LIN {X 0,Y 474.683,Z 210.352,A -85,B 0,C 180,E1 -7368.037,E2 -7368.037} C_VEL
LIN {X 0,Y 474.691,Z 210.355,A -85,B 0,C 180,E1 -7371.486,E2 -7371.486} C_VEL
LIN {X 0,Y 474.74,Z 210.345,A -85,B 0,C 180,E1 -7374.052,E2 -7374.052} C_VEL
LIN {X 0,Y 474.841,Z 210.335,A -85,B 0,C 180,E1 -7377.455,E2 -7377.455} C_VEL
LIN {X 0,Y 474.818,Z 210.341,A -85,B 0,C 180,E1 -7380.848,E2 -7380.848} C_VEL
LIN {X 0,Y 474.835,Z 210.335,A -85,B 0,C 180,E1 -7382.545,E2 -7382.545} C_VEL
LIN {X 0,Y 474.723,Z 210.347,A -85,B 0,C 180,E1 -7385.948,E2 -7385.948} C_VEL
LIN {X 0,Y 474.671,Z 210.356,A -85,B 0,C 180,E1 -7388.515,E2 -7388.515} C_VEL
LIN {X 0,Y 474.683,Z 210.352,A -85,B 0,C 180,E1 -7391.963,E2 -7391.963} C_VEL
LIN {X 0,Y 474.647,Z 210.356,A -85,B 0,C 180,E1 -7395.779,E2 -7395.779} C_VEL
LIN {X 0,Y 474.611,Z 210.365,A -85,B 0,C 180,E1 -7399.013,E2 -7399.013} C_VEL
LIN {X 0,Y 474.545,Z 210.369,A -85,B 0,C 180,E1 -7401.731,E2 -7401.731} C_VEL
LIN {X 0,Y 474.611,Z 210.367,A -85,B 0,C 180,E1 -7404.496,E2 -7404.496} C_VEL
LIN {X 0,Y 474.652,Z 210.356,A -85,B 0,C 180,E1 -7407.342,E2 -7407.342} C_VEL
LIN {X 0,Y 474.565,Z 210.371,A -85,B 0,C 180,E1 -7410.815,E2 -7410.815} C_VEL
LIN {X 0,Y 474.597,Z 210.365,A -85,B 0,C 180,E1 -7413.988,E2 -7413.988} C_VEL
LIN {X 0,Y 474.534,Z 210.372,A -85,B 0,C 180,E1 -7416.903,E2 -7416.903} C_VEL
LIN {X 0,Y 474.611,Z 210.362,A -85,B 0,C 180,E1 -7419.654,E2 -7419.654} C_VEL
LIN {X 0,Y 474.618,Z 210.361,A -85,B 0,C 180,E1 -7422.934,E2 -7422.934} C_VEL
LIN {X 0,Y 474.579,Z 210.368,A -85,B 0,C 180,E1 -7425.899,E2 -7425.899} C_VEL
LIN {X 0,Y 474.601,Z 210.362,A -85,B 0,C 180,E1 -7429.045,E2 -7429.045} C_VEL
LIN {X 0,Y 474.586,Z 210.367,A -85,B 0,C 180,E1 -7431.708,E2 -7431.708} C_VEL
LIN {X 0,Y 474.608,Z 210.362,A -85,B 0,C 180,E1 -7434.73,E2 -7434.73} C_VEL
LIN {X 0,Y 474.617,Z 210.365,A -85,B 0,C 180,E1 -7437.792,E2 -7437.792} C_VEL
LIN {X 0,Y 474.608,Z 210.361,A -85,B 0,C 180,E1 -7440.889,E2 -7440.889} C_VEL
LIN {X 0,Y 474.642,Z 210.361,A -85,B 0,C 180,E1 -7443.632,E2 -7443.632} C_VEL
LIN {X 0,Y 474.625,Z 210.359,A -85,B 0,C 180,E1 -7446.645,E2 -7446.645} C_VEL
LIN {X 0,Y 474.646,Z 210.361,A -85,B 0,C 180,E1 -7450.093,E2 -7450.093} C_VEL
LIN {X 0,Y 474.638,Z 210.362,A -85,B 0,C 180,E1 -7451.71,E2 -7451.71} C_VEL
LIN {X 0,Y 473.972,Z 210.45,A -85,B 0,C 180,E1 -7452.419,E2 -7452.419} C_VEL
LIN {X 0,Y 471.122,Z 210.804,A -85,B 0,C 180,E1 -7453.571,E2 -7453.571} C_VEL
LIN {X 0,Y 468.711,Z 211.1,A -85,B 0,C 180,E1 -7454.5,E2 -7454.5} C_VEL
LIN {X 0,Y 467.673,Z 211.227,A -85,B 0,C 180,E1 -7455.217,E2 -7455.217} C_VEL
LIN {X 0,Y 467.588,Z 211.236,A -85,B 0,C 180,E1 -7455.46,E2 -7455.46} C_VEL
LIN {X 0,Y 467.65,Z 211.232,A -85,B 0,C 180,E1 -7458.737,E2 -7458.737} C_VEL
LIN {X 0,Y 467.708,Z 211.37,A -85,B 0,C 180,E1 -7461.142,E2 -7461.142} C_VEL
LIN {X 0,Y 468.579,Z 217.66,A -85,B 0,C 180,E1 -7462.461,E2 -7462.461} C_VEL
LIN {X 0,Y 468.348,Z 226.062,A -85,B 0,C 180,E1 -7464.135,E2 -7464.135} C_VEL
LIN {X 0,Y 471.304,Z 240.96,A -85,B 0,C 180,E1 -7464.467,E2 -7464.467} C_VEL
LIN {X 0,Y 470.437,Z 333.788,A -85,B 0,C 180,E1 -7465.906,E2 -7465.906} C_VEL
LIN {X 0,Y 470.197,Z 347.368,A -85,B 0,C 180,E1 -7466.306,E2 -7466.306} C_VEL
LIN {X 0,Y 469.865,Z 359.62,A -85,B 0,C 180,E1 -7466.84,E2 -7466.84} C_VEL
LIN {X 0,Y 469.485,Z 371.367,A -85,B 0,C 180,E1 -7467.535,E2 -7467.535} C_VEL
LIN {X 0,Y 468.946,Z 382.682,A -85,B 0,C 180,E1 -7468.392,E2 -7468.392} C_VEL
LIN {X 0,Y 468.486,Z 392.879,A -85,B 0,C 180,E1 -7469.357,E2 -7469.357} C_VEL
LIN {X 0,Y 468.059,Z 402.058,A -85,B 0,C 180,E1 -7470.432,E2 -7470.432} C_VEL
LIN {X 0,Y 467.627,Z 410.968,A -85,B 0,C 180,E1 -7471.724,E2 -7471.724} C_VEL
LIN {X 0,Y 467.285,Z 418.164,A -85,B 0,C 180,E1 -7473.019,E2 -7473.019} C_VEL
LIN {X 0,Y 467.131,Z 423.923,A -85,B 0,C 180,E1 -7474.315,E2 -7474.315} C_VEL
LIN {X 0,Y 466.93,Z 428.479,A -85,B 0,C 180,E1 -7475.616,E2 -7475.616} C_VEL
LIN {X 0,Y 466.819,Z 431.951,A -85,B 0,C 180,E1 -7476.918,E2 -7476.918} C_VEL
LIN {X 0,Y 466.739,Z 433.696,A -85,B 0,C 180,E1 -7477.79,E2 -7477.79} C_VEL
LIN {X 0,Y 466.615,Z 435.959,A -85,B 0,C 180,E1 -7479.537,E2 -7479.537} C_VEL
LIN {X 0,Y 466.637,Z 436.49,A -85,B 0,C 180,E1 -7480.413,E2 -7480.413} C_VEL
LIN {X 0,Y 466.688,Z 436.48,A -85,B 0,C 180,E1 -7481.802,E2 -7481.802} C_VEL
LIN {X 0,Y 466.63,Z 435.592,A -85,B 0,C 180,E1 -7483.057,E2 -7483.057} C_VEL
LIN {X 0,Y 466.66,Z 434.468,A -85,B 0,C 180,E1 -7483.944,E2 -7483.944} C_VEL
LIN {X 0,Y 466.848,Z 431.331,A -85,B 0,C 180,E1 -7485.534,E2 -7485.534} C_VEL
LIN {X 0,Y 466.999,Z 426.929,A -85,B 0,C 180,E1 -7487.065,E2 -7487.065} C_VEL
LIN {X 0,Y 467.242,Z 421.768,A -85,B 0,C 180,E1 -7488.413,E2 -7488.413} C_VEL
LIN {X 0,Y 467.513,Z 415.168,A -85,B 0,C 180,E1 -7489.769,E2 -7489.769} C_VEL
LIN {X 0,Y 468.017,Z 406.854,A -85,B 0,C 180,E1 -7491.124,E2 -7491.124} C_VEL
LIN {X 0,Y 468.456,Z 398.271,A -85,B 0,C 180,E1 -7492.26,E2 -7492.26} C_VEL
LIN {X 0,Y 468.921,Z 388.788,A -85,B 0,C 180,E1 -7493.284,E2 -7493.284} C_VEL
LIN {X 0,Y 469.432,Z 378.914,A -85,B 0,C 180,E1 -7494.148,E2 -7494.148} C_VEL
LIN {X 0,Y 469.92,Z 366.789,A -85,B 0,C 180,E1 -7494.992,E2 -7494.992} C_VEL
LIN {X 0,Y 470.292,Z 354.995,A -85,B 0,C 180,E1 -7495.622,E2 -7495.622} C_VEL
LIN {X 0,Y 470.657,Z 341.985,A -85,B 0,C 180,E1 -7496.114,E2 -7496.114} C_VEL
LIN {X 0,Y 470.883,Z 328.515,A -85,B 0,C 180,E1 -7496.434,E2 -7496.434} C_VEL
LIN {X 0,Y 471.54,Z 239.78,A -85,B 0,C 180,E1 -7497.811,E2 -7497.811} C_VEL
LIN {X 0,Y 468.611,Z 226.016,A -85,B 0,C 180,E1 -7498.174,E2 -7498.174} C_VEL
LIN {X 0,Y 468.575,Z 216.184,A -85,B 0,C 180,E1 -7500.161,E2 -7500.161} C_VEL
LIN {X 0,Y 467.602,Z 211.238,A -85,B 0,C 180,E1 -7501.263,E2 -7501.263} C_VEL
LIN {X 0,Y 467.585,Z 211.242,A -85,B 0,C 180,E1 -7504.241,E2 -7504.241} C_VEL
LIN {X 0,Y 467.544,Z 211.246,A -85,B 0,C 180,E1 -7507.185,E2 -7507.185} C_VEL
LIN {X 0,Y 467.586,Z 211.241,A -85,B 0,C 180,E1 -7510.261,E2 -7510.261} C_VEL
LIN {X 0,Y 467.577,Z 211.243,A -85,B 0,C 180,E1 -7512.565,E2 -7512.565} C_VEL
LIN {X 0,Y 467.562,Z 211.248,A -85,B 0,C 180,E1 -7516.175,E2 -7516.175} C_VEL
LIN {X 0,Y 467.575,Z 211.24,A -85,B 0,C 180,E1 -7518.72,E2 -7518.72} C_VEL
LIN {X 0,Y 467.552,Z 211.247,A -85,B 0,C 180,E1 -7521.954,E2 -7521.954} C_VEL
LIN {X 0,Y 467.548,Z 211.241,A -85,B 0,C 180,E1 -7525.166,E2 -7525.166} C_VEL
LIN {X 0,Y 467.563,Z 211.24,A -85,B 0,C 180,E1 -7528.258,E2 -7528.258} C_VEL
LIN {X 0,Y 467.558,Z 211.242,A -85,B 0,C 180,E1 -7531.249,E2 -7531.249} C_VEL
LIN {X 0,Y 467.586,Z 211.24,A -85,B 0,C 180,E1 -7534.158,E2 -7534.158} C_VEL
LIN {X 0,Y 467.553,Z 211.238,A -85,B 0,C 180,E1 -7536.994,E2 -7536.994} C_VEL
LIN {X 0,Y 467.595,Z 211.237,A -85,B 0,C 180,E1 -7539.776,E2 -7539.776} C_VEL
LIN {X 0,Y 467.583,Z 211.237,A -85,B 0,C 180,E1 -7542.506,E2 -7542.506} C_VEL
LIN {X 0,Y 467.575,Z 211.238,A -85,B 0,C 180,E1 -7545.195,E2 -7545.195} C_VEL
LIN {X 0,Y 467.625,Z 211.233,A -85,B 0,C 180,E1 -7547.854,E2 -7547.854} C_VEL
LIN {X 0,Y 467.651,Z 211.236,A -85,B 0,C 180,E1 -7551.357,E2 -7551.357} C_VEL
LIN {X 0,Y 467.723,Z 211.218,A -85,B 0,C 180,E1 -7553.962,E2 -7553.962} C_VEL
LIN {X 0,Y 467.825,Z 211.208,A -85,B 0,C 180,E1 -7557.417,E2 -7557.417} C_VEL
LIN {X 0,Y 467.844,Z 211.204,A -85,B 0,C 180,E1 -7560,E2 -7560} C_VEL
LIN {X 0,Y 467.823,Z 211.206,A -85,B 0,C 180,E1 -7562.583,E2 -7562.583} C_VEL
LIN {X 0,Y 467.695,Z 211.222,A -85,B 0,C 180,E1 -7566.038,E2 -7566.038} C_VEL
LIN {X 0,Y 467.638,Z 211.229,A -85,B 0,C 180,E1 -7568.644,E2 -7568.644} C_VEL
LIN {X 0,Y 467.643,Z 211.226,A -85,B 0,C 180,E1 -7572.146,E2 -7572.146} C_VEL
LIN {X 0,Y 467.618,Z 211.231,A -85,B 0,C 180,E1 -7575.885,E2 -7575.885} C_VEL
LIN {X 0,Y 467.592,Z 211.238,A -85,B 0,C 180,E1 -7579.309,E2 -7579.309} C_VEL
LIN {X 0,Y 467.502,Z 211.244,A -85,B 0,C 180,E1 -7582.075,E2 -7582.075} C_VEL
LIN {X 0,Y 467.543,Z 211.243,A -85,B 0,C 180,E1 -7584.891,E2 -7584.891} C_VEL
LIN {X 0,Y 467.555,Z 211.241,A -85,B 0,C 180,E1 -7587.773,E2 -7587.773} C_VEL
LIN {X 0,Y 467.527,Z 211.246,A -85,B 0,C 180,E1 -7591.042,E2 -7591.042} C_VEL
LIN {X 0,Y 467.555,Z 211.242,A -85,B 0,C 180,E1 -7594.242,E2 -7594.242} C_VEL
LIN {X 0,Y 467.526,Z 211.239,A -85,B 0,C 180,E1 -7597.187,E2 -7597.187} C_VEL
LIN {X 0,Y 467.555,Z 211.241,A -85,B 0,C 180,E1 -7600.267,E2 -7600.267} C_VEL
LIN {X 0,Y 467.572,Z 211.242,A -85,B 0,C 180,E1 -7602.569,E2 -7602.569} C_VEL
LIN {X 0,Y 467.551,Z 211.24,A -85,B 0,C 180,E1 -7605.054,E2 -7605.054} C_VEL
LIN {X 0,Y 467.555,Z 211.242,A -85,B 0,C 180,E1 -7608.598,E2 -7608.598} C_VEL
LIN {X 0,Y 467.554,Z 211.243,A -85,B 0,C 180,E1 -7611.957,E2 -7611.957} C_VEL
LIN {X 0,Y 467.558,Z 211.241,A -85,B 0,C 180,E1 -7615.169,E2 -7615.169} C_VEL
LIN {X 0,Y 467.578,Z 211.244,A -85,B 0,C 180,E1 -7618.261,E2 -7618.261} C_VEL
LIN {X 0,Y 467.552,Z 211.245,A -85,B 0,C 180,E1 -7621.25,E2 -7621.25} C_VEL
LIN {X 0,Y 467.622,Z 211.273,A -85,B 0,C 180,E1 -7623.352,E2 -7623.352} C_VEL
LIN {X 0,Y 469.977,Z 223.105,A -85,B 0,C 180,E1 -7625.581,E2 -7625.581} C_VEL
LIN {X 0,Y 469.825,Z 230.597,A -85,B 0,C 180,E1 -7626.88,E2 -7626.88} C_VEL
LIN {X 0,Y 469.021,Z 248.029,A -85,B 0,C 180,E1 -7629.84,E2 -7629.84} C_VEL
LIN {X 0,Y 468.331,Z 266.089,A -85,B 0,C 180,E1 -7632.866,E2 -7632.866} C_VEL
LIN {X 0,Y 471.36,Z 286.814,A -85,B 0,C 180,E1 -7633.329,E2 -7633.329} C_VEL
LIN {X 0,Y 470.641,Z 375.192,A -85,B 0,C 180,E1 -7634.713,E2 -7634.713} C_VEL
LIN {X 0,Y 470.204,Z 389.075,A -85,B 0,C 180,E1 -7635.114,E2 -7635.114} C_VEL
LIN {X 0,Y 469.721,Z 401.519,A -85,B 0,C 180,E1 -7635.652,E2 -7635.652} C_VEL
LIN {X 0,Y 469.208,Z 413.424,A -85,B 0,C 180,E1 -7636.354,E2 -7636.354} C_VEL
LIN {X 0,Y 468.662,Z 425.211,A -85,B 0,C 180,E1 -7637.25,E2 -7637.25} C_VEL
LIN {X 0,Y 468.137,Z 436.204,A -85,B 0,C 180,E1 -7638.306,E2 -7638.306} C_VEL
LIN {X 0,Y 467.673,Z 445.316,A -85,B 0,C 180,E1 -7639.391,E2 -7639.391} C_VEL
LIN {X 0,Y 467.248,Z 454.216,A -85,B 0,C 180,E1 -7640.694,E2 -7640.694} C_VEL
LIN {X 0,Y 466.987,Z 461.379,A -85,B 0,C 180,E1 -7641.997,E2 -7641.997} C_VEL
LIN {X 0,Y 466.831,Z 466.228,A -85,B 0,C 180,E1 -7643.082,E2 -7643.082} C_VEL
LIN {X 0,Y 466.733,Z 470.943,A -85,B 0,C 180,E1 -7644.382,E2 -7644.382} C_VEL
LIN {X 0,Y 466.648,Z 474.545,A -85,B 0,C 180,E1 -7645.68,E2 -7645.68} C_VEL
LIN {X 0,Y 466.691,Z 476.404,A -85,B 0,C 180,E1 -7646.545,E2 -7646.545} C_VEL
LIN {X 0,Y 466.68,Z 477.796,A -85,B 0,C 180,E1 -7647.409,E2 -7647.409} C_VEL
LIN {X 0,Y 466.661,Z 478.792,A -85,B 0,C 180,E1 -7648.273,E2 -7648.273} C_VEL
LIN {X 0,Y 466.624,Z 479.396,A -85,B 0,C 180,E1 -7649.135,E2 -7649.135} C_VEL
LIN {X 0,Y 466.607,Z 479.602,A -85,B 0,C 180,E1 -7649.998,E2 -7649.998} C_VEL
LIN {X 0,Y 466.661,Z 478.761,A -85,B 0,C 180,E1 -7651.724,E2 -7651.724} C_VEL
LIN {X 0,Y 466.679,Z 477.755,A -85,B 0,C 180,E1 -7652.588,E2 -7652.588} C_VEL
LIN {X 0,Y 466.691,Z 476.337,A -85,B 0,C 180,E1 -7653.451,E2 -7653.451} C_VEL
LIN {X 0,Y 466.687,Z 473.368,A -85,B 0,C 180,E1 -7654.749,E2 -7654.749} C_VEL
LIN {X 0,Y 466.743,Z 469.348,A -85,B 0,C 180,E1 -7656.048,E2 -7656.048} C_VEL
LIN {X 0,Y 466.906,Z 463.158,A -85,B 0,C 180,E1 -7657.566,E2 -7657.566} C_VEL
LIN {X 0,Y 467.121,Z 456.401,A -85,B 0,C 180,E1 -7658.869,E2 -7658.869} C_VEL
LIN {X 0,Y 467.448,Z 448.015,A -85,B 0,C 180,E1 -7660.173,E2 -7660.173} C_VEL
LIN {X 0,Y 467.905,Z 439.387,A -85,B 0,C 180,E1 -7661.257,E2 -7661.257} C_VEL
LIN {X 0,Y 468.333,Z 429.269,A -85,B 0,C 180,E1 -7662.295,E2 -7662.295} C_VEL
LIN {X 0,Y 468.864,Z 418.178,A -85,B 0,C 180,E1 -7663.211,E2 -7663.211} C_VEL
LIN {X 0,Y 469.352,Z 406.508,A -85,B 0,C 180,E1 -7663.969,E2 -7663.969} C_VEL
LIN {X 0,Y 469.8,Z 394.374,A -85,B 0,C 180,E1 -7664.564,E2 -7664.564} C_VEL
LIN {X 0,Y 470.189,Z 381.179,A -85,B 0,C 180,E1 -7665.022,E2 -7665.022} C_VEL
LIN {X 0,Y 470.523,Z 368.479,A -85,B 0,C 180,E1 -7665.288,E2 -7665.288} C_VEL
LIN {X 0,Y 470.883,Z 285.054,A -85,B 0,C 180,E1 -7666.568,E2 -7666.568} C_VEL
LIN {X 0,Y 468.204,Z 266.3,A -85,B 0,C 180,E1 -7666.966,E2 -7666.966} C_VEL
LIN {X 0,Y 468.844,Z 248.358,A -85,B 0,C 180,E1 -7669.936,E2 -7669.936} C_VEL
LIN {X 0,Y 469.498,Z 230.626,A -85,B 0,C 180,E1 -7672.9,E2 -7672.9} C_VEL
LIN {X 0,Y 469.801,Z 223.259,A -85,B 0,C 180,E1 -7674.142,E2 -7674.142} C_VEL
LIN {X 0,Y 467.665,Z 211.233,A -85,B 0,C 180,E1 -7676.311,E2 -7676.311} C_VEL
LIN {X 0,Y 467.554,Z 211.243,A -85,B 0,C 180,E1 -7679.329,E2 -7679.329} C_VEL
LIN {X 0,Y 467.563,Z 211.24,A -85,B 0,C 180,E1 -7682.675,E2 -7682.675} C_VEL
LIN {X 0,Y 467.541,Z 211.246,A -85,B 0,C 180,E1 -7685.736,E2 -7685.736} C_VEL
LIN {X 0,Y 467.556,Z 211.24,A -85,B 0,C 180,E1 -7689.141,E2 -7689.141} C_VEL
LIN {X 0,Y 467.558,Z 211.24,A -85,B 0,C 180,E1 -7692.563,E2 -7692.563} C_VEL
LIN {X 0,Y 467.541,Z 211.245,A -85,B 0,C 180,E1 -7696.173,E2 -7696.173} C_VEL
LIN {X 0,Y 467.556,Z 211.24,A -85,B 0,C 180,E1 -7698.718,E2 -7698.718} C_VEL
LIN {X 0,Y 467.541,Z 211.245,A -85,B 0,C 180,E1 -7701.403,E2 -7701.403} C_VEL
LIN {X 0,Y 467.522,Z 211.245,A -85,B 0,C 180,E1 -7704.257,E2 -7704.257} C_VEL
LIN {X 0,Y 467.54,Z 211.246,A -85,B 0,C 180,E1 -7707.317,E2 -7707.317} C_VEL
LIN {X 0,Y 467.532,Z 211.243,A -85,B 0,C 180,E1 -7710.663,E2 -7710.663} C_VEL
LIN {X 0,Y 467.572,Z 211.242,A -85,B 0,C 180,E1 -7713.197,E2 -7713.197} C_VEL
LIN {X 0,Y 467.537,Z 211.243,A -85,B 0,C 180,E1 -7716.055,E2 -7716.055} C_VEL
LIN {X 0,Y 467.605,Z 211.235,A -85,B 0,C 180,E1 -7718.856,E2 -7718.856} C_VEL
LIN {X 0,Y 467.58,Z 211.242,A -85,B 0,C 180,E1 -7721.6,E2 -7721.6} C_VEL
LIN {X 0,Y 467.6,Z 211.234,A -85,B 0,C 180,E1 -7724.304,E2 -7724.304} C_VEL
LIN {X 0,Y 467.641,Z 211.23,A -85,B 0,C 180,E1 -7727.854,E2 -7727.854} C_VEL
LIN {X 0,Y 467.64,Z 211.235,A -85,B 0,C 180,E1 -7731.357,E2 -7731.357} C_VEL
LIN {X 0,Y 467.704,Z 211.221,A -85,B 0,C 180,E1 -7733.962,E2 -7733.962} C_VEL
LIN {X 0,Y 467.808,Z 211.212,A -85,B 0,C 180,E1 -7737.417,E2 -7737.417} C_VEL
LIN {X 0,Y 467.77,Z 211.219,A -85,B 0,C 180,E1 -7740.861,E2 -7740.861} C_VEL
LIN {X 0,Y 467.801,Z 211.212,A -85,B 0,C 180,E1 -7742.583,E2 -7742.583} C_VEL
LIN {X 0,Y 467.687,Z 211.223,A -85,B 0,C 180,E1 -7746.038,E2 -7746.038} C_VEL
LIN {X 0,Y 467.626,Z 211.236,A -85,B 0,C 180,E1 -7748.644,E2 -7748.644} C_VEL
LIN {X 0,Y 467.642,Z 211.23,A -85,B 0,C 180,E1 -7752.146,E2 -7752.146} C_VEL
LIN {X 0,Y 467.612,Z 211.233,A -85,B 0,C 180,E1 -7755.894,E2 -7755.894} C_VEL
LIN {X 0,Y 467.57,Z 211.239,A -85,B 0,C 180,E1 -7759.31,E2 -7759.31} C_VEL
LIN {X 0,Y 467.49,Z 211.249,A -85,B 0,C 180,E1 -7762.076,E2 -7762.076} C_VEL
LIN {X 0,Y 467.556,Z 211.244,A -85,B 0,C 180,E1 -7764.89,E2 -7764.89} C_VEL
LIN {X 0,Y 467.582,Z 211.237,A -85,B 0,C 180,E1 -7767.772,E2 -7767.772} C_VEL
LIN {X 0,Y 467.528,Z 211.245,A -85,B 0,C 180,E1 -7771.049,E2 -7771.049} C_VEL
LIN {X 0,Y 467.549,Z 211.246,A -85,B 0,C 180,E1 -7774.246,E2 -7774.246} C_VEL
LIN {X 0,Y 467.51,Z 211.246,A -85,B 0,C 180,E1 -7777.19,E2 -7777.19} C_VEL
LIN {X 0,Y 467.56,Z 211.246,A -85,B 0,C 180,E1 -7780.267,E2 -7780.267} C_VEL
LIN {X 0,Y 467.587,Z 211.24,A -85,B 0,C 180,E1 -7782.575,E2 -7782.575} C_VEL
LIN {X 0,Y 467.539,Z 211.242,A -85,B 0,C 180,E1 -7785.057,E2 -7785.057} C_VEL
LIN {X 0,Y 467.561,Z 211.239,A -85,B 0,C 180,E1 -7787.444,E2 -7787.444} C_VEL
LIN {X 0,Y 467.557,Z 211.24,A -85,B 0,C 180,E1 -7790.859,E2 -7790.859} C_VEL
LIN {X 0,Y 467.541,Z 211.247,A -85,B 0,C 180,E1 -7794.265,E2 -7794.265} C_VEL
LIN {X 0,Y 467.564,Z 211.239,A -85,B 0,C 180,E1 -7797.325,E2 -7797.325} C_VEL
LIN {X 0,Y 467.554,Z 211.241,A -85,B 0,C 180,E1 -7800.672,E2 -7800.672} C_VEL
LIN {X 0,Y 467.6,Z 211.235,A -85,B 0,C 180,E1 -7803.203,E2 -7803.203} C_VEL
LIN {X 0,Y 467.581,Z 211.238,A -85,B 0,C 180,E1 -7806.473,E2 -7806.473} C_VEL
LIN {X 0,Y 467.615,Z 211.24,A -85,B 0,C 180,E1 -7809.781,E2 -7809.781} C_VEL
LIN {X 0,Y 467.589,Z 211.236,A -85,B 0,C 180,E1 -7812.509,E2 -7812.509} C_VEL
LIN {X 0,Y 467.598,Z 211.236,A -85,B 0,C 180,E1 -7815.199,E2 -7815.199} C_VEL
LIN {X 0,Y 467.588,Z 211.236,A -85,B 0,C 180,E1 -7815.46,E2 -7815.46} C_VEL
LIN {X 0,Y 466.92,Z 211.322,A -85,B 0,C 180,E1 -7816.179,E2 -7816.179} C_VEL
LIN {X 0,Y 464.078,Z 211.676,A -85,B 0,C 180,E1 -7817.347,E2 -7817.347} C_VEL
LIN {X 0,Y 461.679,Z 211.977,A -85,B 0,C 180,E1 -7818.29,E2 -7818.29} C_VEL
LIN {X 0,Y 460.653,Z 212.104,A -85,B 0,C 180,E1 -7819.017,E2 -7819.017} C_VEL
LIN {X 0,Y 460.572,Z 212.116,A -85,B 0,C 180,E1 -7819.264,E2 -7819.264} C_VEL
LIN {X 0,Y 460.688,Z 212.281,A -85,B 0,C 180,E1 -7821.006,E2 -7821.006} C_VEL
LIN {X 0,Y 461.591,Z 218.621,A -85,B 0,C 180,E1 -7822.347,E2 -7822.347} C_VEL
LIN {X 0,Y 461.337,Z 226.288,A -85,B 0,C 180,E1 -7823.894,E2 -7823.894} C_VEL
LIN {X 0,Y 464.465,Z 241.723,A -85,B 0,C 180,E1 -7824.249,E2 -7824.249} C_VEL
LIN {X 0,Y 463.534,Z 333.33,A -85,B 0,C 180,E1 -7825.682,E2 -7825.682} C_VEL
LIN {X 0,Y 463.293,Z 346.426,A -85,B 0,C 180,E1 -7826.061,E2 -7826.061} C_VEL
LIN {X 0,Y 462.966,Z 359.563,A -85,B 0,C 180,E1 -7826.63,E2 -7826.63} C_VEL
LIN {X 0,Y 462.634,Z 370.625,A -85,B 0,C 180,E1 -7827.281,E2 -7827.281} C_VEL
LIN {X 0,Y 462.027,Z 382.152,A -85,B 0,C 180,E1 -7828.149,E2 -7828.149} C_VEL
LIN {X 0,Y 461.534,Z 392.502,A -85,B 0,C 180,E1 -7829.129,E2 -7829.129} C_VEL
LIN {X 0,Y 461.071,Z 401.844,A -85,B 0,C 180,E1 -7830.22,E2 -7830.22} C_VEL
LIN {X 0,Y 460.629,Z 410.85,A -85,B 0,C 180,E1 -7831.531,E2 -7831.531} C_VEL
LIN {X 0,Y 460.271,Z 418.125,A -85,B 0,C 180,E1 -7832.846,E2 -7832.846} C_VEL
LIN {X 0,Y 460.054,Z 424.805,A -85,B 0,C 180,E1 -7834.382,E2 -7834.382} C_VEL
LIN {X 0,Y 459.862,Z 429.232,A -85,B 0,C 180,E1 -7835.702,E2 -7835.702} C_VEL
LIN {X 0,Y 459.72,Z 432.596,A -85,B 0,C 180,E1 -7837.026,E2 -7837.026} C_VEL
LIN {X 0,Y 459.64,Z 434.27,A -85,B 0,C 180,E1 -7837.911,E2 -7837.911} C_VEL
LIN {X 0,Y 459.555,Z 435.544,A -85,B 0,C 180,E1 -7838.798,E2 -7838.798} C_VEL
LIN {X 0,Y 459.521,Z 436.418,A -85,B 0,C 180,E1 -7839.686,E2 -7839.686} C_VEL
LIN {X 0,Y 459.571,Z 436.846,A -85,B 0,C 180,E1 -7840.575,E2 -7840.575} C_VEL
LIN {X 0,Y 459.595,Z 436.8,A -85,B 0,C 180,E1 -7841.853,E2 -7841.853} C_VEL
LIN {X 0,Y 459.561,Z 435.768,A -85,B 0,C 180,E1 -7843.262,E2 -7843.262} C_VEL
LIN {X 0,Y 459.589,Z 434.547,A -85,B 0,C 180,E1 -7844.163,E2 -7844.163} C_VEL
LIN {X 0,Y 459.782,Z 431.633,A -85,B 0,C 180,E1 -7845.636,E2 -7845.636} C_VEL
LIN {X 0,Y 459.928,Z 428.222,A -85,B 0,C 180,E1 -7846.878,E2 -7846.878} C_VEL
LIN {X 0,Y 460.154,Z 423.33,A -85,B 0,C 180,E1 -7848.246,E2 -7848.246} C_VEL
LIN {X 0,Y 460.481,Z 417.083,A -85,B 0,C 180,E1 -7849.619,E2 -7849.619} C_VEL
LIN {X 0,Y 460.924,Z 409.223,A -85,B 0,C 180,E1 -7850.997,E2 -7850.997} C_VEL
LIN {X 0,Y 461.412,Z 400.974,A -85,B 0,C 180,E1 -7852.158,E2 -7852.158} C_VEL
LIN {X 0,Y 461.93,Z 391.002,A -85,B 0,C 180,E1 -7853.301,E2 -7853.301} C_VEL
LIN {X 0,Y 462.504,Z 380.705,A -85,B 0,C 180,E1 -7854.253,E2 -7854.253} C_VEL
LIN {X 0,Y 463.021,Z 369.396,A -85,B 0,C 180,E1 -7855.084,E2 -7855.084} C_VEL
LIN {X 0,Y 463.453,Z 356.95,A -85,B 0,C 180,E1 -7855.786,E2 -7855.786} C_VEL
LIN {X 0,Y 463.827,Z 344.429,A -85,B 0,C 180,E1 -7856.3,E2 -7856.3} C_VEL
LIN {X 0,Y 464.024,Z 332.562,A -85,B 0,C 180,E1 -7856.624,E2 -7856.624} C_VEL
LIN {X 0,Y 464.87,Z 241.026,A -85,B 0,C 180,E1 -7858.072,E2 -7858.072} C_VEL
LIN {X 0,Y 461.679,Z 226.379,A -85,B 0,C 180,E1 -7858.459,E2 -7858.459} C_VEL
LIN {X 0,Y 461.703,Z 218.082,A -85,B 0,C 180,E1 -7860.152,E2 -7860.152} C_VEL
LIN {X 0,Y 460.561,Z 212.115,A -85,B 0,C 180,E1 -7861.472,E2 -7861.472} C_VEL
LIN {X 0,Y 460.529,Z 212.122,A -85,B 0,C 180,E1 -7864.504,E2 -7864.504} C_VEL
LIN {X 0,Y 460.523,Z 212.121,A -85,B 0,C 180,E1 -7867.619,E2 -7867.619} C_VEL
LIN {X 0,Y 460.549,Z 212.117,A -85,B 0,C 180,E1 -7870.27,E2 -7870.27} C_VEL
LIN {X 0,Y 460.489,Z 212.123,A -85,B 0,C 180,E1 -7873.374,E2 -7873.374} C_VEL
LIN {X 0,Y 460.512,Z 212.121,A -85,B 0,C 180,E1 -7876.626,E2 -7876.626} C_VEL
LIN {X 0,Y 460.543,Z 212.119,A -85,B 0,C 180,E1 -7879.726,E2 -7879.726} C_VEL
LIN {X 0,Y 460.51,Z 212.119,A -85,B 0,C 180,E1 -7882.518,E2 -7882.518} C_VEL
LIN {X 0,Y 460.529,Z 212.119,A -85,B 0,C 180,E1 -7885.622,E2 -7885.622} C_VEL
LIN {X 0,Y 460.517,Z 212.115,A -85,B 0,C 180,E1 -7888.743,E2 -7888.743} C_VEL
LIN {X 0,Y 460.532,Z 212.12,A -85,B 0,C 180,E1 -7891.765,E2 -7891.765} C_VEL
LIN {X 0,Y 460.535,Z 212.115,A -85,B 0,C 180,E1 -7894.704,E2 -7894.704} C_VEL
LIN {X 0,Y 460.489,Z 212.124,A -85,B 0,C 180,E1 -7897.57,E2 -7897.57} C_VEL
LIN {X 0,Y 460.541,Z 212.111,A -85,B 0,C 180,E1 -7900.383,E2 -7900.383} C_VEL
LIN {X 0,Y 460.595,Z 212.106,A -85,B 0,C 180,E1 -7903.992,E2 -7903.992} C_VEL
LIN {X 0,Y 460.578,Z 212.113,A -85,B 0,C 180,E1 -7907.665,E2 -7907.665} C_VEL
LIN {X 0,Y 460.598,Z 212.112,A -85,B 0,C 180,E1 -7911.223,E2 -7911.223} C_VEL
LIN {X 0,Y 460.69,Z 212.095,A -85,B 0,C 180,E1 -7913.87,E2 -7913.87} C_VEL
LIN {X 0,Y 460.766,Z 212.088,A -85,B 0,C 180,E1 -7917.377,E2 -7917.377} C_VEL
LIN {X 0,Y 460.816,Z 212.08,A -85,B 0,C 180,E1 -7920,E2 -7920} C_VEL
LIN {X 0,Y 460.765,Z 212.086,A -85,B 0,C 180,E1 -7922.623,E2 -7922.623} C_VEL
LIN {X 0,Y 460.66,Z 212.099,A -85,B 0,C 180,E1 -7926.131,E2 -7926.131} C_VEL
LIN {X 0,Y 460.589,Z 212.108,A -85,B 0,C 180,E1 -7928.777,E2 -7928.777} C_VEL
LIN {X 0,Y 460.605,Z 212.105,A -85,B 0,C 180,E1 -7932.458,E2 -7932.458} C_VEL
LIN {X 0,Y 460.572,Z 212.109,A -85,B 0,C 180,E1 -7935.999,E2 -7935.999} C_VEL
LIN {X 0,Y 460.538,Z 212.114,A -85,B 0,C 180,E1 -7939.617,E2 -7939.617} C_VEL
LIN {X 0,Y 460.479,Z 212.122,A -85,B 0,C 180,E1 -7942.43,E2 -7942.43} C_VEL
LIN {X 0,Y 460.522,Z 212.112,A -85,B 0,C 180,E1 -7945.798,E2 -7945.798} C_VEL
LIN {X 0,Y 460.502,Z 212.123,A -85,B 0,C 180,E1 -7948.236,E2 -7948.236} C_VEL
LIN {X 0,Y 460.498,Z 212.12,A -85,B 0,C 180,E1 -7951.284,E2 -7951.284} C_VEL
LIN {X 0,Y 460.501,Z 212.124,A -85,B 0,C 180,E1 -7954.505,E2 -7954.505} C_VEL
LIN {X 0,Y 460.481,Z 212.116,A -85,B 0,C 180,E1 -7957.625,E2 -7957.625} C_VEL
LIN {X 0,Y 460.519,Z 212.117,A -85,B 0,C 180,E1 -7960.27,E2 -7960.27} C_VEL
LIN {X 0,Y 460.481,Z 212.122,A -85,B 0,C 180,E1 -7963.378,E2 -7963.378} C_VEL
LIN {X 0,Y 460.496,Z 212.123,A -85,B 0,C 180,E1 -7966.627,E2 -7966.627} C_VEL
LIN {X 0,Y 460.514,Z 212.12,A -85,B 0,C 180,E1 -7969.735,E2 -7969.735} C_VEL
LIN {X 0,Y 460.491,Z 212.125,A -85,B 0,C 180,E1 -7972.526,E2 -7972.526} C_VEL
LIN {X 0,Y 460.54,Z 212.118,A -85,B 0,C 180,E1 -7975.625,E2 -7975.625} C_VEL
LIN {X 0,Y 460.533,Z 212.119,A -85,B 0,C 180,E1 -7978.746,E2 -7978.746} C_VEL
LIN {X 0,Y 460.548,Z 212.117,A -85,B 0,C 180,E1 -7982.262,E2 -7982.262} C_VEL
LIN {X 0,Y 460.57,Z 212.168,A -85,B 0,C 180,E1 -7983.095,E2 -7983.095} C_VEL
LIN {X 0,Y 463.151,Z 225.067,A -85,B 0,C 180,E1 -7985.569,E2 -7985.569} C_VEL
LIN {X 0,Y 462.511,Z 240.565,A -85,B 0,C 180,E1 -7988.271,E2 -7988.271} C_VEL
LIN {X 0,Y 461.573,Z 261.27,A -85,B 0,C 180,E1 -7991.812,E2 -7991.812} C_VEL
LIN {X 0,Y 461.362,Z 265.823,A -85,B 0,C 180,E1 -7992.583,E2 -7992.583} C_VEL
LIN {X 0,Y 464.606,Z 287.362,A -85,B 0,C 180,E1 -7993.065,E2 -7993.065} C_VEL
LIN {X 0,Y 463.86,Z 374.754,A -85,B 0,C 180,E1 -7994.455,E2 -7994.455} C_VEL
LIN {X 0,Y 463.45,Z 387.903,A -85,B 0,C 180,E1 -7994.836,E2 -7994.836} C_VEL
LIN {X 0,Y 462.92,Z 400.568,A -85,B 0,C 180,E1 -7995.38,E2 -7995.38} C_VEL
LIN {X 0,Y 462.395,Z 411.849,A -85,B 0,C 180,E1 -7996.037,E2 -7996.037} C_VEL
LIN {X 0,Y 461.827,Z 423.223,A -85,B 0,C 180,E1 -7996.892,E2 -7996.892} C_VEL
LIN {X 0,Y 461.291,Z 434.013,A -85,B 0,C 180,E1 -7997.907,E2 -7997.907} C_VEL
LIN {X 0,Y 460.756,Z 443.501,A -85,B 0,C 180,E1 -7999.008,E2 -7999.008} C_VEL
LIN {X 0,Y 460.289,Z 452.652,A -85,B 0,C 180,E1 -8000.33,E2 -8000.33} C_VEL
LIN {X 0,Y 459.971,Z 460.039,A -85,B 0,C 180,E1 -8001.653,E2 -8001.653} C_VEL
LIN {X 0,Y 459.743,Z 465.977,A -85,B 0,C 180,E1 -8002.974,E2 -8002.974} C_VEL
LIN {X 0,Y 459.635,Z 470.673,A -85,B 0,C 180,E1 -8004.295,E2 -8004.295} C_VEL
LIN {X 0,Y 459.566,Z 474.261,A -85,B 0,C 180,E1 -8005.613,E2 -8005.613} C_VEL
LIN {X 0,Y 459.588,Z 476.105,A -85,B 0,C 180,E1 -8006.492,E2 -8006.492} C_VEL
LIN {X 0,Y 459.601,Z 477.491,A -85,B 0,C 180,E1 -8007.369,E2 -8007.369} C_VEL
LIN {X 0,Y 459.557,Z 479.08,A -85,B 0,C 180,E1 -8009.122,E2 -8009.122} C_VEL
LIN {X 0,Y 459.538,Z 479.274,A -85,B 0,C 180,E1 -8009.998,E2 -8009.998} C_VEL
LIN {X 0,Y 459.557,Z 479.04,A -85,B 0,C 180,E1 -8010.875,E2 -8010.875} C_VEL
LIN {X 0,Y 459.6,Z 477.406,A -85,B 0,C 180,E1 -8012.627,E2 -8012.627} C_VEL
LIN {X 0,Y 459.588,Z 475.975,A -85,B 0,C 180,E1 -8013.505,E2 -8013.505} C_VEL
LIN {X 0,Y 459.617,Z 472.994,A -85,B 0,C 180,E1 -8014.822,E2 -8014.822} C_VEL
LIN {X 0,Y 459.712,Z 467.903,A -85,B 0,C 180,E1 -8016.429,E2 -8016.429} C_VEL
LIN {X 0,Y 459.87,Z 461.723,A -85,B 0,C 180,E1 -8017.903,E2 -8017.903} C_VEL
LIN {X 0,Y 460.133,Z 454.709,A -85,B 0,C 180,E1 -8019.226,E2 -8019.226} C_VEL
LIN {X 0,Y 460.504,Z 445.908,A -85,B 0,C 180,E1 -8020.55,E2 -8020.55} C_VEL
LIN {X 0,Y 461.056,Z 435.915,A -85,B 0,C 180,E1 -8021.761,E2 -8021.761} C_VEL
LIN {X 0,Y 461.558,Z 425.128,A -85,B 0,C 180,E1 -8022.806,E2 -8022.806} C_VEL
LIN {X 0,Y 462.072,Z 412.854,A -85,B 0,C 180,E1 -8023.745,E2 -8023.745} C_VEL
LIN {X 0,Y 462.651,Z 400.66,A -85,B 0,C 180,E1 -8024.456,E2 -8024.456} C_VEL
LIN {X 0,Y 463.104,Z 387.83,A -85,B 0,C 180,E1 -8025.004,E2 -8025.004} C_VEL
LIN {X 0,Y 463.495,Z 374.414,A -85,B 0,C 180,E1 -8025.385,E2 -8025.385} C_VEL
LIN {X 0,Y 464.139,Z 287.052,A -85,B 0,C 180,E1 -8026.754,E2 -8026.754} C_VEL
LIN {X 0,Y 461.21,Z 266.056,A -85,B 0,C 180,E1 -8027.19,E2 -8027.19} C_VEL
LIN {X 0,Y 461.829,Z 249.216,A -85,B 0,C 180,E1 -8030.019,E2 -8030.019} C_VEL
LIN {X 0,Y 462.511,Z 232.845,A -85,B 0,C 180,E1 -8032.794,E2 -8032.794} C_VEL
LIN {X 0,Y 462.792,Z 223.871,A -85,B 0,C 180,E1 -8034.333,E2 -8034.333} C_VEL
LIN {X 0,Y 460.642,Z 212.107,A -85,B 0,C 180,E1 -8036.5,E2 -8036.5} C_VEL
LIN {X 0,Y 460.515,Z 212.122,A -85,B 0,C 180,E1 -8039.554,E2 -8039.554} C_VEL
LIN {X 0,Y 460.513,Z 212.122,A -85,B 0,C 180,E1 -8042.28,E2 -8042.28} C_VEL
LIN {X 0,Y 460.492,Z 212.121,A -85,B 0,C 180,E1 -8045.441,E2 -8045.441} C_VEL
LIN {X 0,Y 460.519,Z 212.116,A -85,B 0,C 180,E1 -8048.893,E2 -8048.893} C_VEL
LIN {X 0,Y 460.494,Z 212.123,A -85,B 0,C 180,E1 -8052.177,E2 -8052.177} C_VEL
LIN {X 0,Y 460.49,Z 212.123,A -85,B 0,C 180,E1 -8055.408,E2 -8055.408} C_VEL
LIN {X 0,Y 460.512,Z 212.118,A -85,B 0,C 180,E1 -8058.392,E2 -8058.392} C_VEL
LIN {X 0,Y 460.511,Z 212.12,A -85,B 0,C 180,E1 -8061.265,E2 -8061.265} C_VEL
LIN {X 0,Y 460.472,Z 212.122,A -85,B 0,C 180,E1 -8064.551,E2 -8064.551} C_VEL
LIN {X 0,Y 460.49,Z 212.127,A -85,B 0,C 180,E1 -8067.712,E2 -8067.712} C_VEL
LIN {X 0,Y 460.501,Z 212.119,A -85,B 0,C 180,E1 -8070.766,E2 -8070.766} C_VEL
LIN {X 0,Y 460.52,Z 212.121,A -85,B 0,C 180,E1 -8073.732,E2 -8073.732} C_VEL
LIN {X 0,Y 460.511,Z 212.117,A -85,B 0,C 180,E1 -8076.622,E2 -8076.622} C_VEL
LIN {X 0,Y 460.536,Z 212.122,A -85,B 0,C 180,E1 -8079.452,E2 -8079.452} C_VEL
LIN {X 0,Y 460.508,Z 212.118,A -85,B 0,C 180,E1 -8082.228,E2 -8082.228} C_VEL
LIN {X 0,Y 460.517,Z 212.12,A -85,B 0,C 180,E1 -8084.963,E2 -8084.963} C_VEL
LIN {X 0,Y 460.603,Z 212.109,A -85,B 0,C 180,E1 -8087.666,E2 -8087.666} C_VEL
LIN {X 0,Y 460.608,Z 212.113,A -85,B 0,C 180,E1 -8091.224,E2 -8091.224} C_VEL
LIN {X 0,Y 460.67,Z 212.098,A -85,B 0,C 180,E1 -8093.87,E2 -8093.87} C_VEL
LIN {X 0,Y 460.773,Z 212.089,A -85,B 0,C 180,E1 -8097.377,E2 -8097.377} C_VEL
LIN {X 0,Y 460.792,Z 212.082,A -85,B 0,C 180,E1 -8100,E2 -8100} C_VEL
LIN {X 0,Y 460.742,Z 212.092,A -85,B 0,C 180,E1 -8102.623,E2 -8102.623} C_VEL
LIN {X 0,Y 460.652,Z 212.1,A -85,B 0,C 180,E1 -8106.131,E2 -8106.131} C_VEL
LIN {X 0,Y 460.573,Z 212.116,A -85,B 0,C 180,E1 -8108.777,E2 -8108.777} C_VEL
LIN {X 0,Y 460.58,Z 212.112,A -85,B 0,C 180,E1 -8112.458,E2 -8112.458} C_VEL
LIN {X 0,Y 460.569,Z 212.11,A -85,B 0,C 180,E1 -8116.009,E2 -8116.009} C_VEL
LIN {X 0,Y 460.516,Z 212.117,A -85,B 0,C 180,E1 -8119.618,E2 -8119.618} C_VEL
LIN {X 0,Y 460.465,Z 212.128,A -85,B 0,C 180,E1 -8122.431,E2 -8122.431} C_VEL
LIN {X 0,Y 460.521,Z 212.116,A -85,B 0,C 180,E1 -8125.805,E2 -8125.805} C_VEL
LIN {X 0,Y 460.513,Z 212.121,A -85,B 0,C 180,E1 -8128.236,E2 -8128.236} C_VEL
LIN {X 0,Y 460.48,Z 212.121,A -85,B 0,C 180,E1 -8131.287,E2 -8131.287} C_VEL
LIN {X 0,Y 460.493,Z 212.127,A -85,B 0,C 180,E1 -8134.509,E2 -8134.509} C_VEL
LIN {X 0,Y 460.465,Z 212.123,A -85,B 0,C 180,E1 -8137.627,E2 -8137.627} C_VEL
LIN {X 0,Y 460.522,Z 212.123,A -85,B 0,C 180,E1 -8140.276,E2 -8140.276} C_VEL
LIN {X 0,Y 460.492,Z 212.12,A -85,B 0,C 180,E1 -8143.377,E2 -8143.377} C_VEL
LIN {X 0,Y 460.47,Z 212.125,A -85,B 0,C 180,E1 -8146.629,E2 -8146.629} C_VEL
LIN {X 0,Y 460.516,Z 212.119,A -85,B 0,C 180,E1 -8149.735,E2 -8149.735} C_VEL
LIN {X 0,Y 460.477,Z 212.124,A -85,B 0,C 180,E1 -8152.528,E2 -8152.528} C_VEL
LIN {X 0,Y 460.528,Z 212.118,A -85,B 0,C 180,E1 -8155.628,E2 -8155.628} C_VEL
LIN {X 0,Y 460.521,Z 212.117,A -85,B 0,C 180,E1 -8158.749,E2 -8158.749} C_VEL
LIN {X 0,Y 460.568,Z 212.114,A -85,B 0,C 180,E1 -8162.258,E2 -8162.258} C_VEL
LIN {X 0,Y 460.528,Z 212.115,A -85,B 0,C 180,E1 -8164.708,E2 -8164.708} C_VEL
LIN {X 0,Y 460.502,Z 212.123,A -85,B 0,C 180,E1 -8167.575,E2 -8167.575} C_VEL
LIN {X 0,Y 460.561,Z 212.112,A -85,B 0,C 180,E1 -8170.388,E2 -8170.388} C_VEL
LIN {X 0,Y 460.601,Z 212.11,A -85,B 0,C 180,E1 -8174.062,E2 -8174.062} C_VEL
LIN {X 0,Y 460.608,Z 212.113,A -85,B 0,C 180,E1 -8177.669,E2 -8177.669} C_VEL
LIN {X 0,Y 460.572,Z 212.116,A -85,B 0,C 180,E1 -8179.264,E2 -8179.264} C_VEL
LIN {X 0,Y 459.922,Z 212.296,A -85,B 0,C 180,E1 -8179.76,E2 -8179.76} C_VEL
LIN {X 0,Y 457.234,Z 213.336,A -85,B 0,C 180,E1 -8180.536,E2 -8180.536} C_VEL
LIN {X 0,Y 455.102,Z 214.907,A -85,B 0,C 180,E1 -8181.136,E2 -8181.136} C_VEL
LIN {X 0,Y 454.338,Z 216.58,A -85,B 0,C 180,E1 -8181.586,E2 -8181.586} C_VEL
LIN {X 0,Y 454.366,Z 217.233,A -85,B 0,C 180,E1 -8181.733,E2 -8181.733} C_VEL
LIN {X 0,Y 454.597,Z 222.831,A -85,B 0,C 180,E1 -8182.898,E2 -8182.898} C_VEL
LIN {X 0,Y 454.412,Z 226.775,A -85,B 0,C 180,E1 -8183.662,E2 -8183.662} C_VEL
LIN {X 0,Y 457.562,Z 242.415,A -85,B 0,C 180,E1 -8184.024,E2 -8184.024} C_VEL
LIN {X 0,Y 456.67,Z 333.837,A -85,B 0,C 180,E1 -8185.478,E2 -8185.478} C_VEL
LIN {X 0,Y 456.394,Z 346.89,A -85,B 0,C 180,E1 -8185.863,E2 -8185.863} C_VEL
LIN {X 0,Y 456.073,Z 359.436,A -85,B 0,C 180,E1 -8186.413,E2 -8186.413} C_VEL
LIN {X 0,Y 455.685,Z 371.42,A -85,B 0,C 180,E1 -8187.129,E2 -8187.129} C_VEL
LIN {X 0,Y 455.057,Z 382.865,A -85,B 0,C 180,E1 -8188.01,E2 -8188.01} C_VEL
LIN {X 0,Y 454.549,Z 393.148,A -85,B 0,C 180,E1 -8189.005,E2 -8189.005} C_VEL
LIN {X 0,Y 454.121,Z 401.567,A -85,B 0,C 180,E1 -8190.002,E2 -8190.002} C_VEL
LIN {X 0,Y 453.676,Z 409.354,A -85,B 0,C 180,E1 -8191.111,E2 -8191.111} C_VEL
LIN {X 0,Y 453.255,Z 416.972,A -85,B 0,C 180,E1 -8192.445,E2 -8192.445} C_VEL
LIN {X 0,Y 453.03,Z 423.979,A -85,B 0,C 180,E1 -8194.004,E2 -8194.004} C_VEL
LIN {X 0,Y 452.78,Z 428.669,A -85,B 0,C 180,E1 -8195.345,E2 -8195.345} C_VEL
LIN {X 0,Y 452.7,Z 431.794,A -85,B 0,C 180,E1 -8196.495,E2 -8196.495} C_VEL
LIN {X 0,Y 452.535,Z 434.839,A -85,B 0,C 180,E1 -8198.036,E2 -8198.036} C_VEL
LIN {X 0,Y 452.463,Z 436.058,A -85,B 0,C 180,E1 -8198.937,E2 -8198.937} C_VEL
LIN {X 0,Y 452.432,Z 436.833,A -85,B 0,C 180,E1 -8199.839,E2 -8199.839} C_VEL
LIN {X 0,Y 452.476,Z 437.202,A -85,B 0,C 180,E1 -8200.743,E2 -8200.743} C_VEL
LIN {X 0,Y 452.517,Z 437.115,A -85,B 0,C 180,E1 -8201.916,E2 -8201.916} C_VEL
LIN {X 0,Y 452.471,Z 435.91,A -85,B 0,C 180,E1 -8203.473,E2 -8203.473} C_VEL
LIN {X 0,Y 452.536,Z 434.631,A -85,B 0,C 180,E1 -8204.388,E2 -8204.388} C_VEL
LIN {X 0,Y 452.736,Z 431.922,A -85,B 0,C 180,E1 -8205.75,E2 -8205.75} C_VEL
LIN {X 0,Y 452.877,Z 428.069,A -85,B 0,C 180,E1 -8207.149,E2 -8207.149} C_VEL
LIN {X 0,Y 453.172,Z 423.146,A -85,B 0,C 180,E1 -8208.512,E2 -8208.512} C_VEL
LIN {X 0,Y 453.483,Z 416.653,A -85,B 0,C 180,E1 -8209.935,E2 -8209.935} C_VEL
LIN {X 0,Y 454.043,Z 408.55,A -85,B 0,C 180,E1 -8211.33,E2 -8211.33} C_VEL
LIN {X 0,Y 454.565,Z 400.193,A -85,B 0,C 180,E1 -8212.498,E2 -8212.498} C_VEL
LIN {X 0,Y 455.134,Z 389.886,A -85,B 0,C 180,E1 -8213.67,E2 -8213.67} C_VEL
LIN {X 0,Y 455.742,Z 379.56,A -85,B 0,C 180,E1 -8214.605,E2 -8214.605} C_VEL
LIN {X 0,Y 456.268,Z 368.177,A -85,B 0,C 180,E1 -8215.426,E2 -8215.426} C_VEL
LIN {X 0,Y 456.666,Z 356.592,A -85,B 0,C 180,E1 -8216.076,E2 -8216.076} C_VEL
LIN {X 0,Y 457.085,Z 344.477,A -85,B 0,C 180,E1 -8216.571,E2 -8216.571} C_VEL
LIN {X 0,Y 457.312,Z 331.328,A -85,B 0,C 180,E1 -8216.919,E2 -8216.919} C_VEL
LIN {X 0,Y 458.177,Z 242.174,A -85,B 0,C 180,E1 -8218.348,E2 -8218.348} C_VEL
LIN {X 0,Y 454.785,Z 226.622,A -85,B 0,C 180,E1 -8218.78,E2 -8218.78} C_VEL
LIN {X 0,Y 454.777,Z 219.396,A -85,B 0,C 180,E1 -8220.276,E2 -8220.276} C_VEL
LIN {X 0,Y 453.525,Z 212.991,A -85,B 0,C 180,E1 -8221.708,E2 -8221.708} C_VEL
LIN {X 0,Y 453.477,Z 212.999,A -85,B 0,C 180,E1 -8224.988,E2 -8224.988} C_VEL
LIN {X 0,Y 453.474,Z 213.003,A -85,B 0,C 180,E1 -8228.308,E2 -8228.308} C_VEL
LIN {X 0,Y 453.508,Z 212.995,A -85,B 0,C 180,E1 -8230.605,E2 -8230.605} C_VEL
LIN {X 0,Y 453.454,Z 212.998,A -85,B 0,C 180,E1 -8234.219,E2 -8234.219} C_VEL
LIN {X 0,Y 453.479,Z 212.995,A -85,B 0,C 180,E1 -8237.007,E2 -8237.007} C_VEL
LIN {X 0,Y 453.513,Z 212.993,A -85,B 0,C 180,E1 -8240.552,E2 -8240.552} C_VEL
LIN {X 0,Y 453.438,Z 213.005,A -85,B 0,C 180,E1 -8243.915,E2 -8243.915} C_VEL
LIN {X 0,Y 453.463,Z 212.997,A -85,B 0,C 180,E1 -8247.149,E2 -8247.149} C_VEL
LIN {X 0,Y 453.494,Z 212.995,A -85,B 0,C 180,E1 -8250.269,E2 -8250.269} C_VEL
LIN {X 0,Y 453.482,Z 212.992,A -85,B 0,C 180,E1 -8253.292,E2 -8253.292} C_VEL
LIN {X 0,Y 453.479,Z 212.992,A -85,B 0,C 180,E1 -8256.237,E2 -8256.237} C_VEL
LIN {X 0,Y 453.457,Z 212.998,A -85,B 0,C 180,E1 -8259.116,E2 -8259.116} C_VEL
LIN {X 0,Y 453.485,Z 212.997,A -85,B 0,C 180,E1 -8261.943,E2 -8261.943} C_VEL
LIN {X 0,Y 453.515,Z 212.985,A -85,B 0,C 180,E1 -8264.725,E2 -8264.725} C_VEL
LIN {X 0,Y 453.53,Z 212.985,A -85,B 0,C 180,E1 -8268.378,E2 -8268.378} C_VEL
LIN {X 0,Y 453.623,Z 212.977,A -85,B 0,C 180,E1 -8271.985,E2 -8271.985} C_VEL
LIN {X 0,Y 453.644,Z 212.972,A -85,B 0,C 180,E1 -8274.666,E2 -8274.666} C_VEL
LIN {X 0,Y 453.711,Z 212.967,A -85,B 0,C 180,E1 -8277.336,E2 -8277.336} C_VEL
LIN {X 0,Y 453.787,Z 212.956,A -85,B 0,C 180,E1 -8280,E2 -8280} C_VEL
LIN {X 0,Y 453.709,Z 212.965,A -85,B 0,C 180,E1 -8282.663,E2 -8282.663} C_VEL
LIN {X 0,Y 453.626,Z 212.975,A -85,B 0,C 180,E1 -8286.226,E2 -8286.226} C_VEL
LIN {X 0,Y 453.555,Z 212.986,A -85,B 0,C 180,E1 -8288.914,E2 -8288.914} C_VEL
LIN {X 0,Y 453.552,Z 212.984,A -85,B 0,C 180,E1 -8292.539,E2 -8292.539} C_VEL
LIN {X 0,Y 453.516,Z 212.989,A -85,B 0,C 180,E1 -8296.197,E2 -8296.197} C_VEL
LIN {X 0,Y 453.49,Z 212.997,A -85,B 0,C 180,E1 -8299.04,E2 -8299.04} C_VEL
LIN {X 0,Y 453.448,Z 212.994,A -85,B 0,C 180,E1 -8301.838,E2 -8301.838} C_VEL
LIN {X 0,Y 453.468,Z 212.998,A -85,B 0,C 180,E1 -8304.737,E2 -8304.737} C_VEL
LIN {X 0,Y 453.466,Z 212.997,A -85,B 0,C 180,E1 -8307.951,E2 -8307.951} C_VEL
LIN {X 0,Y 453.436,Z 213.005,A -85,B 0,C 180,E1 -8310.763,E2 -8310.763} C_VEL
LIN {X 0,Y 453.445,Z 212.996,A -85,B 0,C 180,E1 -8313.915,E2 -8313.915} C_VEL
LIN {X 0,Y 453.432,Z 212.994,A -85,B 0,C 180,E1 -8317.192,E2 -8317.192} C_VEL
LIN {X 0,Y 453.478,Z 212.999,A -85,B 0,C 180,E1 -8320.611,E2 -8320.611} C_VEL
LIN {X 0,Y 453.447,Z 213.005,A -85,B 0,C 180,E1 -8324.223,E2 -8324.223} C_VEL
LIN {X 0,Y 453.436,Z 212.999,A -85,B 0,C 180,E1 -8327.005,E2 -8327.005} C_VEL
LIN {X 0,Y 453.461,Z 212.996,A -85,B 0,C 180,E1 -8329.414,E2 -8329.414} C_VEL
LIN {X 0,Y 453.444,Z 213.001,A -85,B 0,C 180,E1 -8332.812,E2 -8332.812} C_VEL
LIN {X 0,Y 453.471,Z 213.002,A -85,B 0,C 180,E1 -8336.089,E2 -8336.089} C_VEL
LIN {X 0,Y 453.471,Z 212.999,A -85,B 0,C 180,E1 -8339.242,E2 -8339.242} C_VEL
LIN {X 0,Y 453.506,Z 212.994,A -85,B 0,C 180,E1 -8342.297,E2 -8342.297} C_VEL
LIN {X 0,Y 453.526,Z 213.079,A -85,B 0,C 180,E1 -8342.829,E2 -8342.829} C_VEL
LIN {X 0,Y 456.02,Z 225.125,A -85,B 0,C 180,E1 -8345.193,E2 -8345.193} C_VEL
LIN {X 0,Y 456.233,Z 229.01,A -85,B 0,C 180,E1 -8345.908,E2 -8345.908} C_VEL
LIN {X 0,Y 455.37,Z 245.066,A -85,B 0,C 180,E1 -8348.735,E2 -8348.735} C_VEL
LIN {X 0,Y 454.575,Z 262.459,A -85,B 0,C 180,E1 -8351.755,E2 -8351.755} C_VEL
LIN {X 0,Y 454.441,Z 265.427,A -85,B 0,C 180,E1 -8352.266,E2 -8352.266} C_VEL
LIN {X 0,Y 457.878,Z 287.849,A -85,B 0,C 180,E1 -8352.792,E2 -8352.792} C_VEL
LIN {X 0,Y 457.097,Z 374.439,A -85,B 0,C 180,E1 -8354.191,E2 -8354.191} C_VEL
LIN {X 0,Y 456.667,Z 387.574,A -85,B 0,C 180,E1 -8354.576,E2 -8354.576} C_VEL
LIN {X 0,Y 456.095,Z 399.67,A -85,B 0,C 180,E1 -8355.099,E2 -8355.099} C_VEL
LIN {X 0,Y 455.494,Z 411.905,A -85,B 0,C 180,E1 -8355.821,E2 -8355.821} C_VEL
LIN {X 0,Y 454.857,Z 424.017,A -85,B 0,C 180,E1 -8356.759,E2 -8356.759} C_VEL
LIN {X 0,Y 454.329,Z 433.931,A -85,B 0,C 180,E1 -8357.719,E2 -8357.719} C_VEL
LIN {X 0,Y 453.775,Z 443.361,A -85,B 0,C 180,E1 -8358.837,E2 -8358.837} C_VEL
LIN {X 0,Y 453.264,Z 452.47,A -85,B 0,C 180,E1 -8360.179,E2 -8360.179} C_VEL
LIN {X 0,Y 452.929,Z 459.828,A -85,B 0,C 180,E1 -8361.522,E2 -8361.522} C_VEL
LIN {X 0,Y 452.67,Z 465.741,A -85,B 0,C 180,E1 -8362.864,E2 -8362.864} C_VEL
LIN {X 0,Y 452.538,Z 470.415,A -85,B 0,C 180,E1 -8364.205,E2 -8364.205} C_VEL
LIN {X 0,Y 452.487,Z 473.985,A -85,B 0,C 180,E1 -8365.545,E2 -8365.545} C_VEL
LIN {X 0,Y 452.485,Z 475.812,A -85,B 0,C 180,E1 -8366.437,E2 -8366.437} C_VEL
LIN {X 0,Y 452.523,Z 477.191,A -85,B 0,C 180,E1 -8367.328,E2 -8367.328} C_VEL
LIN {X 0,Y 452.491,Z 478.765,A -85,B 0,C 180,E1 -8369.108,E2 -8369.108} C_VEL
LIN {X 0,Y 452.471,Z 478.945,A -85,B 0,C 180,E1 -8369.998,E2 -8369.998} C_VEL
LIN {X 0,Y 452.491,Z 478.703,A -85,B 0,C 180,E1 -8370.888,E2 -8370.888} C_VEL
LIN {X 0,Y 452.522,Z 477.053,A -85,B 0,C 180,E1 -8372.669,E2 -8372.669} C_VEL
LIN {X 0,Y 452.488,Z 475.604,A -85,B 0,C 180,E1 -8373.56,E2 -8373.56} C_VEL
LIN {X 0,Y 452.547,Z 472.61,A -85,B 0,C 180,E1 -8374.898,E2 -8374.898} C_VEL
LIN {X 0,Y 452.608,Z 467.99,A -85,B 0,C 180,E1 -8376.394,E2 -8376.394} C_VEL
LIN {X 0,Y 452.821,Z 461.29,A -85,B 0,C 180,E1 -8378.027,E2 -8378.027} C_VEL
LIN {X 0,Y 453.085,Z 454.241,A -85,B 0,C 180,E1 -8379.371,E2 -8379.371} C_VEL
LIN {X 0,Y 453.492,Z 445.402,A -85,B 0,C 180,E1 -8380.715,E2 -8380.715} C_VEL
LIN {X 0,Y 454.044,Z 435.366,A -85,B 0,C 180,E1 -8381.945,E2 -8381.945} C_VEL
LIN {X 0,Y 454.569,Z 424.5,A -85,B 0,C 180,E1 -8383.006,E2 -8383.006} C_VEL
LIN {X 0,Y 455.05,Z 413.745,A -85,B 0,C 180,E1 -8383.847,E2 -8383.847} C_VEL
LIN {X 0,Y 455.654,Z 401.957,A -85,B 0,C 180,E1 -8384.569,E2 -8384.569} C_VEL
LIN {X 0,Y 456.165,Z 389.063,A -85,B 0,C 180,E1 -8385.152,E2 -8385.152} C_VEL
LIN {X 0,Y 456.519,Z 376.411,A -85,B 0,C 180,E1 -8385.54,E2 -8385.54} C_VEL
LIN {X 0,Y 456.791,Z 357.348,A -85,B 0,C 180,E1 -8385.874,E2 -8385.874} C_VEL
LIN {X 0,Y 457.182,Z 286.489,A -85,B 0,C 180,E1 -8386.992,E2 -8386.992} C_VEL
LIN {X 0,Y 454.214,Z 265.775,A -85,B 0,C 180,E1 -8387.425,E2 -8387.425} C_VEL
LIN {X 0,Y 454.844,Z 248.692,A -85,B 0,C 180,E1 -8390.34,E2 -8390.34} C_VEL
LIN {X 0,Y 455.571,Z 232.309,A -85,B 0,C 180,E1 -8393.161,E2 -8393.161} C_VEL
LIN {X 0,Y 455.866,Z 225.248,A -85,B 0,C 180,E1 -8394.388,E2 -8394.388} C_VEL
LIN {X 0,Y 453.607,Z 212.984,A -85,B 0,C 180,E1 -8396.695,E2 -8396.695} C_VEL
LIN {X 0,Y 453.456,Z 213.002,A -85,B 0,C 180,E1 -8399.781,E2 -8399.781} C_VEL
LIN {X 0,Y 453.471,Z 212.994,A -85,B 0,C 180,E1 -8403.185,E2 -8403.185} C_VEL
LIN {X 0,Y 453.433,Z 213.003,A -85,B 0,C 180,E1 -8406.295,E2 -8406.295} C_VEL
LIN {X 0,Y 453.464,Z 212.997,A -85,B 0,C 180,E1 -8409.446,E2 -8409.446} C_VEL
LIN {X 0,Y 453.448,Z 213.005,A -85,B 0,C 180,E1 -8411.931,E2 -8411.931} C_VEL
LIN {X 0,Y 453.461,Z 212.999,A -85,B 0,C 180,E1 -8415.466,E2 -8415.466} C_VEL
LIN {X 0,Y 453.463,Z 212.998,A -85,B 0,C 180,E1 -8418.207,E2 -8418.207} C_VEL
LIN {X 0,Y 453.498,Z 212.991,A -85,B 0,C 180,E1 -8420.783,E2 -8420.783} C_VEL
LIN {X 0,Y 453.417,Z 213.006,A -85,B 0,C 180,E1 -8423.914,E2 -8423.914} C_VEL
LIN {X 0,Y 453.441,Z 213,A -85,B 0,C 180,E1 -8427.148,E2 -8427.148} C_VEL
LIN {X 0,Y 453.47,Z 212.995,A -85,B 0,C 180,E1 -8430.268,E2 -8430.268} C_VEL
LIN {X 0,Y 453.465,Z 213,A -85,B 0,C 180,E1 -8433.291,E2 -8433.291} C_VEL
LIN {X 0,Y 453.467,Z 212.995,A -85,B 0,C 180,E1 -8436.237,E2 -8436.237} C_VEL
LIN {X 0,Y 453.477,Z 212.998,A -85,B 0,C 180,E1 -8439.117,E2 -8439.117} C_VEL
LIN {X 0,Y 453.46,Z 212.997,A -85,B 0,C 180,E1 -8441.942,E2 -8441.942} C_VEL
LIN {X 0,Y 453.497,Z 212.992,A -85,B 0,C 180,E1 -8444.725,E2 -8444.725} C_VEL
LIN {X 0,Y 453.534,Z 212.986,A -85,B 0,C 180,E1 -8448.378,E2 -8448.378} C_VEL
LIN {X 0,Y 453.602,Z 212.978,A -85,B 0,C 180,E1 -8451.984,E2 -8451.984} C_VEL
LIN {X 0,Y 453.624,Z 212.977,A -85,B 0,C 180,E1 -8454.666,E2 -8454.666} C_VEL
LIN {X 0,Y 453.714,Z 212.969,A -85,B 0,C 180,E1 -8457.337,E2 -8457.337} C_VEL
LIN {X 0,Y 453.763,Z 212.958,A -85,B 0,C 180,E1 -8460,E2 -8460} C_VEL
LIN {X 0,Y 453.687,Z 212.971,A -85,B 0,C 180,E1 -8462.664,E2 -8462.664} C_VEL
LIN {X 0,Y 453.619,Z 212.976,A -85,B 0,C 180,E1 -8466.226,E2 -8466.226} C_VEL
LIN {X 0,Y 453.538,Z 212.994,A -85,B 0,C 180,E1 -8468.915,E2 -8468.915} C_VEL
LIN {X 0,Y 453.548,Z 212.989,A -85,B 0,C 180,E1 -8472.552,E2 -8472.552} C_VEL
LIN {X 0,Y 453.504,Z 212.992,A -85,B 0,C 180,E1 -8476.198,E2 -8476.198} C_VEL
LIN {X 0,Y 453.467,Z 212.998,A -85,B 0,C 180,E1 -8479.042,E2 -8479.042} C_VEL
LIN {X 0,Y 453.428,Z 213,A -85,B 0,C 180,E1 -8481.839,E2 -8481.839} C_VEL
LIN {X 0,Y 453.466,Z 213.001,A -85,B 0,C 180,E1 -8484.737,E2 -8484.737} C_VEL
LIN {X 0,Y 453.493,Z 212.993,A -85,B 0,C 180,E1 -8487.964,E2 -8487.964} C_VEL
LIN {X 0,Y 453.44,Z 213.003,A -85,B 0,C 180,E1 -8490.763,E2 -8490.763} C_VEL
LIN {X 0,Y 453.437,Z 213,A -85,B 0,C 180,E1 -8493.916,E2 -8493.916} C_VEL
LIN {X 0,Y 453.415,Z 213.001,A -85,B 0,C 180,E1 -8497.194,E2 -8497.194} C_VEL
LIN {X 0,Y 453.491,Z 212.992,A -85,B 0,C 180,E1 -8499.45,E2 -8499.45} C_VEL
LIN {X 0,Y 453.459,Z 212.996,A -85,B 0,C 180,E1 -8502.996,E2 -8502.996} C_VEL
LIN {X 0,Y 453.436,Z 213.001,A -85,B 0,C 180,E1 -8505.783,E2 -8505.783} C_VEL
LIN {X 0,Y 453.452,Z 213.005,A -85,B 0,C 180,E1 -8508.213,E2 -8508.213} C_VEL
LIN {X 0,Y 453.49,Z 212.993,A -85,B 0,C 180,E1 -8510.794,E2 -8510.794} C_VEL
LIN {X 0,Y 453.435,Z 213.004,A -85,B 0,C 180,E1 -8513.922,E2 -8513.922} C_VEL
LIN {X 0,Y 453.465,Z 212.995,A -85,B 0,C 180,E1 -8517.155,E2 -8517.155} C_VEL
LIN {X 0,Y 453.459,Z 213,A -85,B 0,C 180,E1 -8520.272,E2 -8520.272} C_VEL
LIN {X 0,Y 453.489,Z 212.993,A -85,B 0,C 180,E1 -8523.298,E2 -8523.298} C_VEL
LIN {X 0,Y 453.488,Z 212.995,A -85,B 0,C 180,E1 -8526.242,E2 -8526.242} C_VEL
LIN {X 0,Y 453.474,Z 212.994,A -85,B 0,C 180,E1 -8529.121,E2 -8529.121} C_VEL
LIN {X 0,Y 453.496,Z 212.997,A -85,B 0,C 180,E1 -8531.948,E2 -8531.948} C_VEL
LIN {X 0,Y 453.534,Z 212.986,A -85,B 0,C 180,E1 -8534.729,E2 -8534.729} C_VEL
LIN {X 0,Y 453.558,Z 212.988,A -85,B 0,C 180,E1 -8538.382,E2 -8538.382} C_VEL
LIN {X 0,Y 453.625,Z 213.086,A -85,B 0,C 180,E1 -8540.837,E2 -8540.837} C_VEL
LIN {X 0,Y 454.366,Z 217.233,A -85,B 0,C 180,E1 -8541.733,E2 -8541.733} C_VEL
LIN {X 0,Y 453.9,Z 219.539,A -85,B 0,C 180,E1 -8542.184,E2 -8542.184} C_VEL
LIN {X 0,Y 450.911,Z 223.613,A -85,B 0,C 180,E1 -8542.884,E2 -8542.884} C_VEL
LIN {X 0,Y 448.911,Z 227.234,A -85,B 0,C 180,E1 -8543.274,E2 -8543.274} C_VEL
LIN {X 0,Y 448.318,Z 230.112,A -85,B 0,C 180,E1 -8543.465,E2 -8543.465} C_VEL
LIN {X 0,Y 448.489,Z 231.986,A -85,B 0,C 180,E1 -8543.535,E2 -8543.535} C_VEL
LIN {X 0,Y 450.737,Z 244.573,A -85,B 0,C 180,E1 -8543.82,E2 -8543.82} C_VEL
LIN {X 0,Y 449.805,Z 334.249,A -85,B 0,C 180,E1 -8545.269,E2 -8545.269} C_VEL
LIN {X 0,Y 449.493,Z 347.29,A -85,B 0,C 180,E1 -8545.659,E2 -8545.659} C_VEL
LIN {X 0,Y 449.182,Z 359.26,A -85,B 0,C 180,E1 -8546.189,E2 -8546.189} C_VEL
LIN {X 0,Y 448.813,Z 370.581,A -85,B 0,C 180,E1 -8546.86,E2 -8546.86} C_VEL
LIN {X 0,Y 448.153,Z 382.268,A -85,B 0,C 180,E1 -8547.755,E2 -8547.755} C_VEL
LIN {X 0,Y 447.615,Z 392.712,A -85,B 0,C 180,E1 -8548.765,E2 -8548.765} C_VEL
LIN {X 0,Y 447.137,Z 401.266,A -85,B 0,C 180,E1 -8549.777,E2 -8549.777} C_VEL
LIN {X 0,Y 446.699,Z 409.154,A -85,B 0,C 180,E1 -8550.903,E2 -8550.903} C_VEL
LIN {X 0,Y 446.229,Z 416.906,A -85,B 0,C 180,E1 -8552.258,E2 -8552.258} C_VEL
LIN {X 0,Y 446.019,Z 423.09,A -85,B 0,C 180,E1 -8553.615,E2 -8553.615} C_VEL
LIN {X 0,Y 445.732,Z 428.038,A -85,B 0,C 180,E1 -8554.976,E2 -8554.976} C_VEL
LIN {X 0,Y 445.62,Z 432.207,A -85,B 0,C 180,E1 -8556.488,E2 -8556.488} C_VEL
LIN {X 0,Y 445.449,Z 435.403,A -85,B 0,C 180,E1 -8558.164,E2 -8558.164} C_VEL
LIN {X 0,Y 445.383,Z 436.533,A -85,B 0,C 180,E1 -8559.08,E2 -8559.08} C_VEL
LIN {X 0,Y 445.385,Z 437.557,A -85,B 0,C 180,E1 -8560.916,E2 -8560.916} C_VEL
LIN {X 0,Y 445.431,Z 437.434,A -85,B 0,C 180,E1 -8561.974,E2 -8561.974} C_VEL
LIN {X 0,Y 445.407,Z 436.053,A -85,B 0,C 180,E1 -8563.691,E2 -8563.691} C_VEL
LIN {X 0,Y 445.498,Z 434.721,A -85,B 0,C 180,E1 -8564.62,E2 -8564.62} C_VEL
LIN {X 0,Y 445.664,Z 432.249,A -85,B 0,C 180,E1 -8565.854,E2 -8565.854} C_VEL
LIN {X 0,Y 445.868,Z 427.927,A -85,B 0,C 180,E1 -8567.427,E2 -8567.427} C_VEL
LIN {X 0,Y 446.174,Z 423.186,A -85,B 0,C 180,E1 -8568.734,E2 -8568.734} C_VEL
LIN {X 0,Y 446.481,Z 417.392,A -85,B 0,C 180,E1 -8570.021,E2 -8570.021} C_VEL
LIN {X 0,Y 447.043,Z 409.585,A -85,B 0,C 180,E1 -8571.414,E2 -8571.414} C_VEL
LIN {X 0,Y 447.603,Z 401.181,A -85,B 0,C 180,E1 -8572.624,E2 -8572.624} C_VEL
LIN {X 0,Y 448.209,Z 391.021,A -85,B 0,C 180,E1 -8573.813,E2 -8573.813} C_VEL
LIN {X 0,Y 448.842,Z 381.127,A -85,B 0,C 180,E1 -8574.746,E2 -8574.746} C_VEL
LIN {X 0,Y 449.409,Z 369.854,A -85,B 0,C 180,E1 -8575.594,E2 -8575.594} C_VEL
LIN {X 0,Y 449.895,Z 357.487,A -85,B 0,C 180,E1 -8576.311,E2 -8576.311} C_VEL
LIN {X 0,Y 450.339,Z 344.737,A -85,B 0,C 180,E1 -8576.845,E2 -8576.845} C_VEL
LIN {X 0,Y 450.579,Z 331.75,A -85,B 0,C 180,E1 -8577.194,E2 -8577.194} C_VEL
LIN {X 0,Y 451.51,Z 243.232,A -85,B 0,C 180,E1 -8578.634,E2 -8578.634} C_VEL
LIN {X 0,Y 447.91,Z 226.915,A -85,B 0,C 180,E1 -8579.104,E2 -8579.104} C_VEL
LIN {X 0,Y 447.891,Z 221.013,A -85,B 0,C 180,E1 -8580.342,E2 -8580.342} C_VEL
LIN {X 0,Y 446.466,Z 213.872,A -85,B 0,C 180,E1 -8581.95,E2 -8581.95} C_VEL
LIN {X 0,Y 446.426,Z 213.877,A -85,B 0,C 180,E1 -8585.052,E2 -8585.052} C_VEL
LIN {X 0,Y 446.429,Z 213.88,A -85,B 0,C 180,E1 -8588.081,E2 -8588.081} C_VEL
LIN {X 0,Y 446.435,Z 213.876,A -85,B 0,C 180,E1 -8590.918,E2 -8590.918} C_VEL
LIN {X 0,Y 446.39,Z 213.878,A -85,B 0,C 180,E1 -8593.844,E2 -8593.844} C_VEL
LIN {X 0,Y 446.434,Z 213.877,A -85,B 0,C 180,E1 -8596.395,E2 -8596.395} C_VEL
LIN {X 0,Y 446.453,Z 213.874,A -85,B 0,C 180,E1 -8599.803,E2 -8599.803} C_VEL
LIN {X 0,Y 446.415,Z 213.877,A -85,B 0,C 180,E1 -8602.121,E2 -8602.121} C_VEL
LIN {X 0,Y 446.412,Z 213.877,A -85,B 0,C 180,E1 -8605.475,E2 -8605.475} C_VEL
LIN {X 0,Y 446.398,Z 213.874,A -85,B 0,C 180,E1 -8608.698,E2 -8608.698} C_VEL
LIN {X 0,Y 446.464,Z 213.871,A -85,B 0,C 180,E1 -8611.82,E2 -8611.82} C_VEL
LIN {X 0,Y 446.434,Z 213.872,A -85,B 0,C 180,E1 -8614.846,E2 -8614.846} C_VEL
LIN {X 0,Y 446.424,Z 213.874,A -85,B 0,C 180,E1 -8618.244,E2 -8618.244} C_VEL
LIN {X 0,Y 446.431,Z 213.876,A -85,B 0,C 180,E1 -8621.648,E2 -8621.648} C_VEL
LIN {X 0,Y 446.484,Z 213.861,A -85,B 0,C 180,E1 -8624.479,E2 -8624.479} C_VEL
LIN {X 0,Y 446.488,Z 213.863,A -85,B 0,C 180,E1 -8628.192,E2 -8628.192} C_VEL
LIN {X 0,Y 446.571,Z 213.856,A -85,B 0,C 180,E1 -8631.857,E2 -8631.857} C_VEL
LIN {X 0,Y 446.619,Z 213.846,A -85,B 0,C 180,E1 -8634.582,E2 -8634.582} C_VEL
LIN {X 0,Y 446.63,Z 213.842,A -85,B 0,C 180,E1 -8638.196,E2 -8638.196} C_VEL
LIN {X 0,Y 446.758,Z 213.831,A -85,B 0,C 180,E1 -8640,E2 -8640} C_VEL
LIN {X 0,Y 446.657,Z 213.844,A -85,B 0,C 180,E1 -8642.706,E2 -8642.706} C_VEL
LIN {X 0,Y 446.594,Z 213.851,A -85,B 0,C 180,E1 -8646.324,E2 -8646.324} C_VEL
LIN {X 0,Y 446.503,Z 213.867,A -85,B 0,C 180,E1 -8649.056,E2 -8649.056} C_VEL
LIN {X 0,Y 446.493,Z 213.864,A -85,B 0,C 180,E1 -8652.731,E2 -8652.731} C_VEL
LIN {X 0,Y 446.46,Z 213.87,A -85,B 0,C 180,E1 -8656.46,E2 -8656.46} C_VEL
LIN {X 0,Y 446.441,Z 213.872,A -85,B 0,C 180,E1 -8659.304,E2 -8659.304} C_VEL
LIN {X 0,Y 446.389,Z 213.875,A -85,B 0,C 180,E1 -8662.201,E2 -8662.201} C_VEL
LIN {X 0,Y 446.413,Z 213.872,A -85,B 0,C 180,E1 -8665.155,E2 -8665.155} C_VEL
LIN {X 0,Y 446.418,Z 213.877,A -85,B 0,C 180,E1 -8668.183,E2 -8668.183} C_VEL
LIN {X 0,Y 446.386,Z 213.878,A -85,B 0,C 180,E1 -8671.303,E2 -8671.303} C_VEL
LIN {X 0,Y 446.402,Z 213.88,A -85,B 0,C 180,E1 -8674.526,E2 -8674.526} C_VEL
LIN {X 0,Y 446.393,Z 213.87,A -85,B 0,C 180,E1 -8678.08,E2 -8678.08} C_VEL
LIN {X 0,Y 446.41,Z 213.875,A -85,B 0,C 180,E1 -8681.393,E2 -8681.393} C_VEL
LIN {X 0,Y 446.409,Z 213.875,A -85,B 0,C 180,E1 -8684.894,E2 -8684.894} C_VEL
LIN {X 0,Y 446.408,Z 213.877,A -85,B 0,C 180,E1 -8687.727,E2 -8687.727} C_VEL
LIN {X 0,Y 446.398,Z 213.876,A -85,B 0,C 180,E1 -8690.971,E2 -8690.971} C_VEL
LIN {X 0,Y 446.413,Z 213.876,A -85,B 0,C 180,E1 -8694.375,E2 -8694.375} C_VEL
LIN {X 0,Y 446.417,Z 213.876,A -85,B 0,C 180,E1 -8697.64,E2 -8697.64} C_VEL
LIN {X 0,Y 446.434,Z 213.875,A -85,B 0,C 180,E1 -8700.791,E2 -8700.791} C_VEL
LIN {X 0,Y 446.489,Z 214.008,A -85,B 0,C 180,E1 -8702.556,E2 -8702.556} C_VEL
LIN {X 0,Y 449.2,Z 227.002,A -85,B 0,C 180,E1 -8705.155,E2 -8705.155} C_VEL
LIN {X 0,Y 449.351,Z 230.379,A -85,B 0,C 180,E1 -8705.785,E2 -8705.785} C_VEL
LIN {X 0,Y 448.417,Z 246.284,A -85,B 0,C 180,E1 -8708.63,E2 -8708.63} C_VEL
LIN {X 0,Y 447.579,Z 263.662,A -85,B 0,C 180,E1 -8711.697,E2 -8711.697} C_VEL
LIN {X 0,Y 447.49,Z 265.015,A -85,B 0,C 180,E1 -8711.933,E2 -8711.933} C_VEL
LIN {X 0,Y 450.767,Z 285.786,A -85,B 0,C 180,E1 -8712.447,E2 -8712.447} C_VEL
LIN {X 0,Y 451.109,Z 291.193,A -85,B 0,C 180,E1 -8712.552,E2 -8712.552} C_VEL
LIN {X 0,Y 450.344,Z 374.234,A -85,B 0,C 180,E1 -8713.918,E2 -8713.918} C_VEL
LIN {X 0,Y 449.863,Z 388.079,A -85,B 0,C 180,E1 -8714.337,E2 -8714.337} C_VEL
LIN {X 0,Y 449.265,Z 399.952,A -85,B 0,C 180,E1 -8714.868,E2 -8714.868} C_VEL
LIN {X 0,Y 448.622,Z 411.997,A -85,B 0,C 180,E1 -8715.599,E2 -8715.599} C_VEL
LIN {X 0,Y 447.966,Z 423.746,A -85,B 0,C 180,E1 -8716.527,E2 -8716.527} C_VEL
LIN {X 0,Y 447.374,Z 433.878,A -85,B 0,C 180,E1 -8717.525,E2 -8717.525} C_VEL
LIN {X 0,Y 446.8,Z 443.239,A -85,B 0,C 180,E1 -8718.66,E2 -8718.66} C_VEL
LIN {X 0,Y 446.234,Z 452.306,A -85,B 0,C 180,E1 -8720.023,E2 -8720.023} C_VEL
LIN {X 0,Y 445.865,Z 459.631,A -85,B 0,C 180,E1 -8721.387,E2 -8721.387} C_VEL
LIN {X 0,Y 445.598,Z 465.517,A -85,B 0,C 180,E1 -8722.75,E2 -8722.75} C_VEL
LIN {X 0,Y 445.46,Z 469.706,A -85,B 0,C 180,E1 -8723.967,E2 -8723.967} C_VEL
LIN {X 0,Y 445.413,Z 473.717,A -85,B 0,C 180,E1 -8725.474,E2 -8725.474} C_VEL
LIN {X 0,Y 445.384,Z 475.523,A -85,B 0,C 180,E1 -8726.38,E2 -8726.38} C_VEL
LIN {X 0,Y 445.446,Z 476.894,A -85,B 0,C 180,E1 -8727.286,E2 -8727.286} C_VEL
LIN {X 0,Y 445.398,Z 478.451,A -85,B 0,C 180,E1 -8729.094,E2 -8729.094} C_VEL
LIN {X 0,Y 445.407,Z 478.614,A -85,B 0,C 180,E1 -8729.998,E2 -8729.998} C_VEL
LIN {X 0,Y 445.399,Z 477.724,A -85,B 0,C 180,E1 -8731.807,E2 -8731.807} C_VEL
LIN {X 0,Y 445.446,Z 476.695,A -85,B 0,C 180,E1 -8732.711,E2 -8732.711} C_VEL
LIN {X 0,Y 445.389,Z 475.227,A -85,B 0,C 180,E1 -8733.617,E2 -8733.617} C_VEL
LIN {X 0,Y 445.477,Z 472.216,A -85,B 0,C 180,E1 -8734.976,E2 -8734.976} C_VEL
LIN {X 0,Y 445.527,Z 467.972,A -85,B 0,C 180,E1 -8736.383,E2 -8736.383} C_VEL
LIN {X 0,Y 445.701,Z 461.861,A -85,B 0,C 180,E1 -8737.928,E2 -8737.928} C_VEL
LIN {X 0,Y 445.973,Z 455.025,A -85,B 0,C 180,E1 -8739.293,E2 -8739.293} C_VEL
LIN {X 0,Y 446.372,Z 446.517,A -85,B 0,C 180,E1 -8740.658,E2 -8740.658} C_VEL
LIN {X 0,Y 446.891,Z 437.749,A -85,B 0,C 180,E1 -8741.794,E2 -8741.794} C_VEL
LIN {X 0,Y 447.4,Z 427.677,A -85,B 0,C 180,E1 -8742.861,E2 -8742.861} C_VEL
LIN {X 0,Y 447.996,Z 416.183,A -85,B 0,C 180,E1 -8743.838,E2 -8743.838} C_VEL
LIN {X 0,Y 448.571,Z 404.103,A -85,B 0,C 180,E1 -8744.631,E2 -8744.631} C_VEL
LIN {X 0,Y 449.165,Z 391.52,A -85,B 0,C 180,E1 -8745.249,E2 -8745.249} C_VEL
LIN {X 0,Y 449.555,Z 379.372,A -85,B 0,C 180,E1 -8745.671,E2 -8745.671} C_VEL
LIN {X 0,Y 449.858,Z 365.861,A -85,B 0,C 180,E1 -8745.95,E2 -8745.95} C_VEL
LIN {X 0,Y 450.329,Z 287.234,A -85,B 0,C 180,E1 -8747.209,E2 -8747.209} C_VEL
LIN {X 0,Y 447.212,Z 265.423,A -85,B 0,C 180,E1 -8747.677,E2 -8747.677} C_VEL
LIN {X 0,Y 447.923,Z 248.156,A -85,B 0,C 180,E1 -8750.669,E2 -8750.669} C_VEL
LIN {X 0,Y 448.68,Z 231.762,A -85,B 0,C 180,E1 -8753.538,E2 -8753.538} C_VEL
LIN {X 0,Y 448.918,Z 227.121,A -85,B 0,C 180,E1 -8754.355,E2 -8754.355} C_VEL
LIN {X 0,Y 446.738,Z 214.768,A -85,B 0,C 180,E1 -8756.683,E2 -8756.683} C_VEL
LIN {X 0,Y 446.559,Z 213.861,A -85,B 0,C 180,E1 -8756.923,E2 -8756.923} C_VEL
LIN {X 0,Y 446.411,Z 213.88,A -85,B 0,C 180,E1 -8760.246,E2 -8760.246} C_VEL
LIN {X 0,Y 446.426,Z 213.873,A -85,B 0,C 180,E1 -8763.45,E2 -8763.45} C_VEL
LIN {X 0,Y 446.38,Z 213.878,A -85,B 0,C 180,E1 -8766.741,E2 -8766.741} C_VEL
LIN {X 0,Y 446.417,Z 213.877,A -85,B 0,C 180,E1 -8770.194,E2 -8770.194} C_VEL
LIN {X 0,Y 446.4,Z 213.876,A -85,B 0,C 180,E1 -8772.601,E2 -8772.601} C_VEL
LIN {X 0,Y 446.425,Z 213.872,A -85,B 0,C 180,E1 -8775.099,E2 -8775.099} C_VEL
LIN {X 0,Y 446.41,Z 213.874,A -85,B 0,C 180,E1 -8778.607,E2 -8778.607} C_VEL
LIN {X 0,Y 446.441,Z 213.87,A -85,B 0,C 180,E1 -8780.973,E2 -8780.973} C_VEL
LIN {X 0,Y 446.381,Z 213.878,A -85,B 0,C 180,E1 -8784.37,E2 -8784.37} C_VEL
LIN {X 0,Y 446.381,Z 213.885,A -85,B 0,C 180,E1 -8787.635,E2 -8787.635} C_VEL
LIN {X 0,Y 446.425,Z 213.872,A -85,B 0,C 180,E1 -8790.789,E2 -8790.789} C_VEL
LIN {X 0,Y 446.431,Z 213.875,A -85,B 0,C 180,E1 -8793.845,E2 -8793.845} C_VEL
LIN {X 0,Y 446.398,Z 213.876,A -85,B 0,C 180,E1 -8796.822,E2 -8796.822} C_VEL
LIN {X 0,Y 446.426,Z 213.875,A -85,B 0,C 180,E1 -8799.736,E2 -8799.736} C_VEL
LIN {X 0,Y 446.413,Z 213.874,A -85,B 0,C 180,E1 -8802.595,E2 -8802.595} C_VEL
LIN {X 0,Y 446.424,Z 213.879,A -85,B 0,C 180,E1 -8805.411,E2 -8805.411} C_VEL
LIN {X 0,Y 446.493,Z 213.863,A -85,B 0,C 180,E1 -8808.192,E2 -8808.192} C_VEL
LIN {X 0,Y 446.551,Z 213.857,A -85,B 0,C 180,E1 -8811.857,E2 -8811.857} C_VEL
LIN {X 0,Y 446.599,Z 213.852,A -85,B 0,C 180,E1 -8814.582,E2 -8814.582} C_VEL
LIN {X 0,Y 446.659,Z 213.848,A -85,B 0,C 180,E1 -8817.294,E2 -8817.294} C_VEL
LIN {X 0,Y 446.734,Z 213.833,A -85,B 0,C 180,E1 -8820,E2 -8820} C_VEL
LIN {X 0,Y 446.634,Z 213.85,A -85,B 0,C 180,E1 -8822.706,E2 -8822.706} C_VEL
LIN {X 0,Y 446.589,Z 213.853,A -85,B 0,C 180,E1 -8826.325,E2 -8826.325} C_VEL
LIN {X 0,Y 446.484,Z 213.87,A -85,B 0,C 180,E1 -8829.057,E2 -8829.057} C_VEL
LIN {X 0,Y 446.481,Z 213.872,A -85,B 0,C 180,E1 -8832.731,E2 -8832.731} C_VEL
LIN {X 0,Y 446.444,Z 213.874,A -85,B 0,C 180,E1 -8836.461,E2 -8836.461} C_VEL
LIN {X 0,Y 446.418,Z 213.874,A -85,B 0,C 180,E1 -8839.306,E2 -8839.306} C_VEL
LIN {X 0,Y 446.37,Z 213.881,A -85,B 0,C 180,E1 -8842.202,E2 -8842.202} C_VEL
LIN {X 0,Y 446.41,Z 213.875,A -85,B 0,C 180,E1 -8845.155,E2 -8845.155} C_VEL
LIN {X 0,Y 446.44,Z 213.873,A -85,B 0,C 180,E1 -8848.182,E2 -8848.182} C_VEL
LIN {X 0,Y 446.376,Z 213.878,A -85,B 0,C 180,E1 -8851.304,E2 -8851.304} C_VEL
LIN {X 0,Y 446.39,Z 213.883,A -85,B 0,C 180,E1 -8854.527,E2 -8854.527} C_VEL
LIN {X 0,Y 446.382,Z 213.881,A -85,B 0,C 180,E1 -8858.084,E2 -8858.084} C_VEL
LIN {X 0,Y 446.411,Z 213.875,A -85,B 0,C 180,E1 -8860.924,E2 -8860.924} C_VEL
LIN {X 0,Y 446.414,Z 213.876,A -85,B 0,C 180,E1 -8863.845,E2 -8863.845} C_VEL
LIN {X 0,Y 446.37,Z 213.884,A -85,B 0,C 180,E1 -8866.408,E2 -8866.408} C_VEL
LIN {X 0,Y 446.401,Z 213.875,A -85,B 0,C 180,E1 -8869.087,E2 -8869.087} C_VEL
LIN {X 0,Y 446.392,Z 213.881,A -85,B 0,C 180,E1 -8871.925,E2 -8871.925} C_VEL
LIN {X 0,Y 446.41,Z 213.875,A -85,B 0,C 180,E1 -8875.481,E2 -8875.481} C_VEL
LIN {X 0,Y 446.399,Z 213.876,A -85,B 0,C 180,E1 -8878.704,E2 -8878.704} C_VEL
LIN {X 0,Y 446.472,Z 213.872,A -85,B 0,C 180,E1 -8881.825,E2 -8881.825} C_VEL
LIN {X 0,Y 446.433,Z 213.871,A -85,B 0,C 180,E1 -8884.851,E2 -8884.851} C_VEL
LIN {X 0,Y 446.44,Z 213.873,A -85,B 0,C 180,E1 -8888.249,E2 -8888.249} C_VEL
LIN {X 0,Y 446.445,Z 213.875,A -85,B 0,C 180,E1 -8891.652,E2 -8891.652} C_VEL
LIN {X 0,Y 446.503,Z 213.863,A -85,B 0,C 180,E1 -8894.483,E2 -8894.483} C_VEL
LIN {X 0,Y 446.516,Z 213.867,A -85,B 0,C 180,E1 -8898.196,E2 -8898.196} C_VEL
LIN {X 0,Y 446.569,Z 213.883,A -85,B 0,C 180,E1 -8900.662,E2 -8900.662} C_VEL
LIN {X 0,Y 447.638,Z 220.521,A -85,B 0,C 180,E1 -8902.106,E2 -8902.106} C_VEL
LIN {X 0,Y 447.479,Z 227.07,A -85,B 0,C 180,E1 -8903.418,E2 -8903.418} C_VEL
LIN {X 0,Y 448.489,Z 231.986,A -85,B 0,C 180,E1 -8903.535,E2 -8903.535} C_VEL
LIN {X 0,Y 448.944,Z 235.832,A -85,B 0,C 180,E1 -8903.614,E2 -8903.614} C_VEL
LIN {X 0,Y 448.415,Z 241.698,A -85,B 0,C 180,E1 -8903.691,E2 -8903.691} C_VEL
LIN {X 0,Y 444.056,Z 259.292,A -85,B 0,C 180,E1 -8903.826,E2 -8903.826} C_VEL
LIN {X 0,Y 443.72,Z 263.293,A -85,B 0,C 180,E1 -8903.88,E2 -8903.88} C_VEL
LIN {X 0,Y 442.917,Z 334.593,A -85,B 0,C 180,E1 -8905.053,E2 -8905.053} C_VEL
LIN {X 0,Y 442.595,Z 347.628,A -85,B 0,C 180,E1 -8905.448,E2 -8905.448} C_VEL
LIN {X 0,Y 442.245,Z 360.156,A -85,B 0,C 180,E1 -8906.015,E2 -8906.015} C_VEL
LIN {X 0,Y 441.868,Z 371.329,A -85,B 0,C 180,E1 -8906.697,E2 -8906.697} C_VEL
LIN {X 0,Y 441.18,Z 382.921,A -85,B 0,C 180,E1 -8907.605,E2 -8907.605} C_VEL
LIN {X 0,Y 440.629,Z 393.311,A -85,B 0,C 180,E1 -8908.631,E2 -8908.631} C_VEL
LIN {X 0,Y 440.086,Z 402.697,A -85,B 0,C 180,E1 -8909.773,E2 -8909.773} C_VEL
LIN {X 0,Y 439.551,Z 411.741,A -85,B 0,C 180,E1 -8911.147,E2 -8911.147} C_VEL
LIN {X 0,Y 439.117,Z 419.04,A -85,B 0,C 180,E1 -8912.524,E2 -8912.524} C_VEL
LIN {X 0,Y 438.851,Z 425.741,A -85,B 0,C 180,E1 -8914.134,E2 -8914.134} C_VEL
LIN {X 0,Y 438.642,Z 430.179,A -85,B 0,C 180,E1 -8915.518,E2 -8915.518} C_VEL
LIN {X 0,Y 438.548,Z 432.633,A -85,B 0,C 180,E1 -8916.489,E2 -8916.489} C_VEL
LIN {X 0,Y 438.455,Z 434.449,A -85,B 0,C 180,E1 -8917.368,E2 -8917.368} C_VEL
LIN {X 0,Y 438.347,Z 435.943,A -85,B 0,C 180,E1 -8918.297,E2 -8918.297} C_VEL
LIN {X 0,Y 438.277,Z 437.644,A -85,B 0,C 180,E1 -8920.16,E2 -8920.16} C_VEL
LIN {X 0,Y 438.295,Z 437.912,A -85,B 0,C 180,E1 -8921.095,E2 -8921.095} C_VEL
LIN {X 0,Y 438.339,Z 437.757,A -85,B 0,C 180,E1 -8922.031,E2 -8922.031} C_VEL
LIN {X 0,Y 438.347,Z 436.2,A -85,B 0,C 180,E1 -8923.916,E2 -8923.916} C_VEL
LIN {X 0,Y 438.446,Z 434.811,A -85,B 0,C 180,E1 -8924.861,E2 -8924.861} C_VEL
LIN {X 0,Y 438.616,Z 432.557,A -85,B 0,C 180,E1 -8925.973,E2 -8925.973} C_VEL
LIN {X 0,Y 438.877,Z 427.785,A -85,B 0,C 180,E1 -8927.714,E2 -8927.714} C_VEL
LIN {X 0,Y 439.233,Z 422.004,A -85,B 0,C 180,E1 -8929.258,E2 -8929.258} C_VEL
LIN {X 0,Y 439.752,Z 414.453,A -85,B 0,C 180,E1 -8930.83,E2 -8930.83} C_VEL
LIN {X 0,Y 440.342,Z 406.748,A -85,B 0,C 180,E1 -8932.108,E2 -8932.108} C_VEL
LIN {X 0,Y 440.962,Z 397.455,A -85,B 0,C 180,E1 -8933.356,E2 -8933.356} C_VEL
LIN {X 0,Y 441.565,Z 387.478,A -85,B 0,C 180,E1 -8934.444,E2 -8934.444} C_VEL
LIN {X 0,Y 442.31,Z 376.476,A -85,B 0,C 180,E1 -8935.404,E2 -8935.404} C_VEL
LIN {X 0,Y 442.825,Z 364.964,A -85,B 0,C 180,E1 -8936.193,E2 -8936.193} C_VEL
LIN {X 0,Y 443.348,Z 352.015,A -85,B 0,C 180,E1 -8936.857,E2 -8936.857} C_VEL
LIN {X 0,Y 443.736,Z 339.312,A -85,B 0,C 180,E1 -8937.31,E2 -8937.31} C_VEL
LIN {X 0,Y 443.969,Z 324.019,A -85,B 0,C 180,E1 -8937.624,E2 -8937.624} C_VEL
LIN {X 0,Y 444.778,Z 243.827,A -85,B 0,C 180,E1 -8938.943,E2 -8938.943} C_VEL
LIN {X 0,Y 441.025,Z 227.326,A -85,B 0,C 180,E1 -8939.418,E2 -8939.418} C_VEL
LIN {X 0,Y 440.777,Z 221.468,A -85,B 0,C 180,E1 -8940.678,E2 -8940.678} C_VEL
LIN {X 0,Y 439.417,Z 214.749,A -85,B 0,C 180,E1 -8942.233,E2 -8942.233} C_VEL
LIN {X 0,Y 439.391,Z 214.752,A -85,B 0,C 180,E1 -8945.339,E2 -8945.339} C_VEL
LIN {X 0,Y 439.389,Z 214.758,A -85,B 0,C 180,E1 -8948.592,E2 -8948.592} C_VEL
LIN {X 0,Y 439.39,Z 214.753,A -85,B 0,C 180,E1 -8951.256,E2 -8951.256} C_VEL
LIN {X 0,Y 439.391,Z 214.752,A -85,B 0,C 180,E1 -8954.727,E2 -8954.727} C_VEL
LIN {X 0,Y 439.396,Z 214.752,A -85,B 0,C 180,E1 -8957.795,E2 -8957.795} C_VEL
LIN {X 0,Y 439.434,Z 214.748,A -85,B 0,C 180,E1 -8960.228,E2 -8960.228} C_VEL
LIN {X 0,Y 439.359,Z 214.756,A -85,B 0,C 180,E1 -8963.711,E2 -8963.711} C_VEL
LIN {X 0,Y 439.354,Z 214.754,A -85,B 0,C 180,E1 -8967.052,E2 -8967.052} C_VEL
LIN {X 0,Y 439.374,Z 214.754,A -85,B 0,C 180,E1 -8970.273,E2 -8970.273} C_VEL
LIN {X 0,Y 439.406,Z 214.746,A -85,B 0,C 180,E1 -8973.395,E2 -8973.395} C_VEL
LIN {X 0,Y 439.363,Z 214.749,A -85,B 0,C 180,E1 -8976.428,E2 -8976.428} C_VEL
LIN {X 0,Y 439.363,Z 214.757,A -85,B 0,C 180,E1 -8979.396,E2 -8979.396} C_VEL
LIN {X 0,Y 439.406,Z 214.748,A -85,B 0,C 180,E1 -8982.308,E2 -8982.308} C_VEL
LIN {X 0,Y 439.421,Z 214.744,A -85,B 0,C 180,E1 -8985.173,E2 -8985.173} C_VEL
LIN {X 0,Y 439.455,Z 214.74,A -85,B 0,C 180,E1 -8988,E2 -8988} C_VEL
LIN {X 0,Y 439.519,Z 214.736,A -85,B 0,C 180,E1 -8991.726,E2 -8991.726} C_VEL
LIN {X 0,Y 439.595,Z 214.721,A -85,B 0,C 180,E1 -8994.495,E2 -8994.495} C_VEL
LIN {X 0,Y 439.6,Z 214.717,A -85,B 0,C 180,E1 -8998.168,E2 -8998.168} C_VEL
LIN {X 0,Y 439.728,Z 214.707,A -85,B 0,C 180,E1 -9000,E2 -9000} C_VEL
LIN {X 0,Y 439.607,Z 214.722,A -85,B 0,C 180,E1 -9002.749,E2 -9002.749} C_VEL
LIN {X 0,Y 439.565,Z 214.727,A -85,B 0,C 180,E1 -9006.426,E2 -9006.426} C_VEL
LIN {X 0,Y 439.467,Z 214.744,A -85,B 0,C 180,E1 -9009.202,E2 -9009.202} C_VEL
LIN {X 0,Y 439.465,Z 214.739,A -85,B 0,C 180,E1 -9012.72,E2 -9012.72} C_VEL
LIN {X 0,Y 439.418,Z 214.746,A -85,B 0,C 180,E1 -9016.348,E2 -9016.348} C_VEL
LIN {X 0,Y 439.375,Z 214.751,A -85,B 0,C 180,E1 -9019.628,E2 -9019.628} C_VEL
LIN {X 0,Y 439.335,Z 214.758,A -85,B 0,C 180,E1 -9022.577,E2 -9022.577} C_VEL
LIN {X 0,Y 439.352,Z 214.749,A -85,B 0,C 180,E1 -9025.588,E2 -9025.588} C_VEL
LIN {X 0,Y 439.374,Z 214.754,A -85,B 0,C 180,E1 -9028.677,E2 -9028.677} C_VEL
LIN {X 0,Y 439.341,Z 214.758,A -85,B 0,C 180,E1 -9032.03,E2 -9032.03} C_VEL
LIN {X 0,Y 439.372,Z 214.752,A -85,B 0,C 180,E1 -9035.341,E2 -9035.341} C_VEL
LIN {X 0,Y 439.352,Z 214.745,A -85,B 0,C 180,E1 -9038.598,E2 -9038.598} C_VEL
LIN {X 0,Y 439.371,Z 214.752,A -85,B 0,C 180,E1 -9041.258,E2 -9041.258} C_VEL
LIN {X 0,Y 439.364,Z 214.753,A -85,B 0,C 180,E1 -9044.734,E2 -9044.734} C_VEL
LIN {X 0,Y 439.371,Z 214.753,A -85,B 0,C 180,E1 -9047.795,E2 -9047.795} C_VEL
LIN {X 0,Y 439.353,Z 214.754,A -85,B 0,C 180,E1 -9051.404,E2 -9051.404} C_VEL
LIN {X 0,Y 439.393,Z 214.75,A -85,B 0,C 180,E1 -9054.845,E2 -9054.845} C_VEL
LIN {X 0,Y 439.368,Z 214.758,A -85,B 0,C 180,E1 -9058.141,E2 -9058.141} C_VEL
LIN {X 0,Y 439.401,Z 214.753,A -85,B 0,C 180,E1 -9061.606,E2 -9061.606} C_VEL
LIN {X 0,Y 439.451,Z 214.838,A -85,B 0,C 180,E1 -9062.253,E2 -9062.253} C_VEL
LIN {X 0,Y 442.215,Z 228.017,A -85,B 0,C 180,E1 -9064.943,E2 -9064.943} C_VEL
LIN {X 0,Y 442.418,Z 232.824,A -85,B 0,C 180,E1 -9065.855,E2 -9065.855} C_VEL
LIN {X 0,Y 441.324,Z 250.184,A -85,B 0,C 180,E1 -9069.004,E2 -9069.004} C_VEL
LIN {X 0,Y 440.588,Z 264.696,A -85,B 0,C 180,E1 -9071.605,E2 -9071.605} C_VEL
LIN {X 0,Y 443.854,Z 284.951,A -85,B 0,C 180,E1 -9072.117,E2 -9072.117} C_VEL
LIN {X 0,Y 444.431,Z 291.406,A -85,B 0,C 180,E1 -9072.253,E2 -9072.253} C_VEL
LIN {X 0,Y 443.603,Z 374.13,A -85,B 0,C 180,E1 -9073.638,E2 -9073.638} C_VEL
LIN {X 0,Y 443.089,Z 387.894,A -85,B 0,C 180,E1 -9074.062,E2 -9074.062} C_VEL
LIN {X 0,Y 442.437,Z 400.267,A -85,B 0,C 180,E1 -9074.628,E2 -9074.628} C_VEL
LIN {X 0,Y 441.739,Z 412.126,A -85,B 0,C 180,E1 -9075.37,E2 -9075.37} C_VEL
LIN {X 0,Y 441.03,Z 424.034,A -85,B 0,C 180,E1 -9076.333,E2 -9076.333} C_VEL
LIN {X 0,Y 440.419,Z 433.85,A -85,B 0,C 180,E1 -9077.325,E2 -9077.325} C_VEL
LIN {X 0,Y 439.83,Z 443.134,A -85,B 0,C 180,E1 -9078.478,E2 -9078.478} C_VEL
LIN {X 0,Y 439.188,Z 452.158,A -85,B 0,C 180,E1 -9079.861,E2 -9079.861} C_VEL
LIN {X 0,Y 438.821,Z 459.449,A -85,B 0,C 180,E1 -9081.248,E2 -9081.248} C_VEL
LIN {X 0,Y 438.524,Z 465.304,A -85,B 0,C 180,E1 -9082.633,E2 -9082.633} C_VEL
LIN {X 0,Y 438.36,Z 469.9,A -85,B 0,C 180,E1 -9084.008,E2 -9084.008} C_VEL
LIN {X 0,Y 438.341,Z 473.456,A -85,B 0,C 180,E1 -9085.401,E2 -9085.401} C_VEL
LIN {X 0,Y 438.285,Z 475.24,A -85,B 0,C 180,E1 -9086.321,E2 -9086.321} C_VEL
LIN {X 0,Y 438.371,Z 476.602,A -85,B 0,C 180,E1 -9087.242,E2 -9087.242} C_VEL
LIN {X 0,Y 438.308,Z 478.137,A -85,B 0,C 180,E1 -9089.08,E2 -9089.08} C_VEL
LIN {X 0,Y 438.314,Z 478.282,A -85,B 0,C 180,E1 -9089.998,E2 -9089.998} C_VEL
LIN {X 0,Y 438.318,Z 477.372,A -85,B 0,C 180,E1 -9091.836,E2 -9091.836} C_VEL
LIN {X 0,Y 438.371,Z 476.334,A -85,B 0,C 180,E1 -9092.755,E2 -9092.755} C_VEL
LIN {X 0,Y 438.292,Z 474.843,A -85,B 0,C 180,E1 -9093.675,E2 -9093.675} C_VEL
LIN {X 0,Y 438.406,Z 471.812,A -85,B 0,C 180,E1 -9095.056,E2 -9095.056} C_VEL
LIN {X 0,Y 438.446,Z 467.706,A -85,B 0,C 180,E1 -9096.44,E2 -9096.44} C_VEL
LIN {X 0,Y 438.653,Z 461.402,A -85,B 0,C 180,E1 -9098.056,E2 -9098.056} C_VEL
LIN {X 0,Y 438.91,Z 454.531,A -85,B 0,C 180,E1 -9099.444,E2 -9099.444} C_VEL
LIN {X 0,Y 439.362,Z 445.969,A -85,B 0,C 180,E1 -9100.83,E2 -9100.83} C_VEL
LIN {X 0,Y 439.875,Z 437.152,A -85,B 0,C 180,E1 -9101.985,E2 -9101.985} C_VEL
LIN {X 0,Y 440.504,Z 426.413,A -85,B 0,C 180,E1 -9103.126,E2 -9103.126} C_VEL
LIN {X 0,Y 441.045,Z 415.42,A -85,B 0,C 180,E1 -9104.061,E2 -9104.061} C_VEL
LIN {X 0,Y 441.686,Z 403.209,A -85,B 0,C 180,E1 -9104.864,E2 -9104.864} C_VEL
LIN {X 0,Y 442.29,Z 390.443,A -85,B 0,C 180,E1 -9105.491,E2 -9105.491} C_VEL
LIN {X 0,Y 442.718,Z 377.791,A -85,B 0,C 180,E1 -9105.919,E2 -9105.919} C_VEL
LIN {X 0,Y 442.967,Z 361.639,A -85,B 0,C 180,E1 -9106.235,E2 -9106.235} C_VEL
LIN {X 0,Y 443.485,Z 288.119,A -85,B 0,C 180,E1 -9107.428,E2 -9107.428} C_VEL
LIN {X 0,Y 440.224,Z 265.026,A -85,B 0,C 180,E1 -9107.942,E2 -9107.942} C_VEL
LIN {X 0,Y 441.079,Z 246.25,A -85,B 0,C 180,E1 -9111.249,E2 -9111.249} C_VEL
LIN {X 0,Y 441.932,Z 229.833,A -85,B 0,C 180,E1 -9114.169,E2 -9114.169} C_VEL
LIN {X 0,Y 441.437,Z 224.759,A -85,B 0,C 180,E1 -9115.113,E2 -9115.113} C_VEL
LIN {X 0,Y 439.486,Z 214.742,A -85,B 0,C 180,E1 -9117.077,E2 -9117.077} C_VEL
LIN {X 0,Y 439.364,Z 214.757,A -85,B 0,C 180,E1 -9120.257,E2 -9120.257} C_VEL
LIN {X 0,Y 439.377,Z 214.754,A -85,B 0,C 180,E1 -9123.72,E2 -9123.72} C_VEL
LIN {X 0,Y 439.326,Z 214.756,A -85,B 0,C 180,E1 -9126.883,E2 -9126.883} C_VEL
LIN {X 0,Y 439.376,Z 214.757,A -85,B 0,C 180,E1 -9129.845,E2 -9129.845} C_VEL
LIN {X 0,Y 439.353,Z 214.753,A -85,B 0,C 180,E1 -9132.623,E2 -9132.623} C_VEL
LIN {X 0,Y 439.371,Z 214.756,A -85,B 0,C 180,E1 -9136.03,E2 -9136.03} C_VEL
LIN {X 0,Y 439.366,Z 214.752,A -85,B 0,C 180,E1 -9139.018,E2 -9139.018} C_VEL
LIN {X 0,Y 439.357,Z 214.759,A -85,B 0,C 180,E1 -9141.601,E2 -9141.601} C_VEL
LIN {X 0,Y 439.36,Z 214.752,A -85,B 0,C 180,E1 -9144.84,E2 -9144.84} C_VEL
LIN {X 0,Y 439.332,Z 214.757,A -85,B 0,C 180,E1 -9148.136,E2 -9148.136} C_VEL
LIN {X 0,Y 439.381,Z 214.754,A -85,B 0,C 180,E1 -9151.324,E2 -9151.324} C_VEL
LIN {X 0,Y 439.367,Z 214.751,A -85,B 0,C 180,E1 -9154.413,E2 -9154.413} C_VEL
LIN {X 0,Y 439.338,Z 214.763,A -85,B 0,C 180,E1 -9157.423,E2 -9157.423} C_VEL
LIN {X 0,Y 439.393,Z 214.749,A -85,B 0,C 180,E1 -9160.66,E2 -9160.66} C_VEL
LIN {X 0,Y 439.423,Z 214.744,A -85,B 0,C 180,E1 -9164.223,E2 -9164.223} C_VEL
LIN {X 0,Y 439.459,Z 214.74,A -85,B 0,C 180,E1 -9168.001,E2 -9168.001} C_VEL
LIN {X 0,Y 439.499,Z 214.736,A -85,B 0,C 180,E1 -9171.725,E2 -9171.725} C_VEL
LIN {X 0,Y 439.574,Z 214.726,A -85,B 0,C 180,E1 -9174.495,E2 -9174.495} C_VEL
LIN {X 0,Y 439.579,Z 214.725,A -85,B 0,C 180,E1 -9178.168,E2 -9178.168} C_VEL
LIN {X 0,Y 439.705,Z 214.709,A -85,B 0,C 180,E1 -9180,E2 -9180} C_VEL
LIN {X 0,Y 439.584,Z 214.729,A -85,B 0,C 180,E1 -9182.749,E2 -9182.749} C_VEL
LIN {X 0,Y 439.56,Z 214.729,A -85,B 0,C 180,E1 -9186.426,E2 -9186.426} C_VEL
LIN {X 0,Y 439.447,Z 214.745,A -85,B 0,C 180,E1 -9189.203,E2 -9189.203} C_VEL
LIN {X 0,Y 439.452,Z 214.747,A -85,B 0,C 180,E1 -9192.728,E2 -9192.728} C_VEL
LIN {X 0,Y 439.408,Z 214.749,A -85,B 0,C 180,E1 -9196.356,E2 -9196.356} C_VEL
LIN {X 0,Y 439.352,Z 214.753,A -85,B 0,C 180,E1 -9199.629,E2 -9199.629} C_VEL
LIN {X 0,Y 439.317,Z 214.764,A -85,B 0,C 180,E1 -9202.578,E2 -9202.578} C_VEL
LIN {X 0,Y 439.358,Z 214.752,A -85,B 0,C 180,E1 -9205.588,E2 -9205.588} C_VEL
LIN {X 0,Y 439.381,Z 214.755,A -85,B 0,C 180,E1 -9208.676,E2 -9208.676} C_VEL
LIN {X 0,Y 439.331,Z 214.757,A -85,B 0,C 180,E1 -9211.864,E2 -9211.864} C_VEL
LIN {X 0,Y 439.361,Z 214.753,A -85,B 0,C 180,E1 -9215.16,E2 -9215.16} C_VEL
LIN {X 0,Y 439.353,Z 214.758,A -85,B 0,C 180,E1 -9218.598,E2 -9218.598} C_VEL
LIN {X 0,Y 439.367,Z 214.751,A -85,B 0,C 180,E1 -9221.263,E2 -9221.263} C_VEL
LIN {X 0,Y 439.378,Z 214.752,A -85,B 0,C 180,E1 -9224.733,E2 -9224.733} C_VEL
LIN {X 0,Y 439.369,Z 214.754,A -85,B 0,C 180,E1 -9227.8,E2 -9227.8} C_VEL
LIN {X 0,Y 439.412,Z 214.753,A -85,B 0,C 180,E1 -9230.233,E2 -9230.233} C_VEL
LIN {X 0,Y 439.353,Z 214.756,A -85,B 0,C 180,E1 -9233.717,E2 -9233.717} C_VEL
LIN {X 0,Y 439.354,Z 214.753,A -85,B 0,C 180,E1 -9237.058,E2 -9237.058} C_VEL
LIN {X 0,Y 439.367,Z 214.755,A -85,B 0,C 180,E1 -9240.278,E2 -9240.278} C_VEL
LIN {X 0,Y 439.416,Z 214.747,A -85,B 0,C 180,E1 -9243.4,E2 -9243.4} C_VEL
LIN {X 0,Y 439.374,Z 214.752,A -85,B 0,C 180,E1 -9246.433,E2 -9246.433} C_VEL
LIN {X 0,Y 439.38,Z 214.752,A -85,B 0,C 180,E1 -9249.401,E2 -9249.401} C_VEL
LIN {X 0,Y 439.399,Z 214.749,A -85,B 0,C 180,E1 -9252.312,E2 -9252.312} C_VEL
LIN {X 0,Y 439.442,Z 214.743,A -85,B 0,C 180,E1 -9255.177,E2 -9255.177} C_VEL
LIN {X 0,Y 439.482,Z 214.744,A -85,B 0,C 180,E1 -9258.004,E2 -9258.004} C_VEL
LIN {X 0,Y 439.534,Z 214.814,A -85,B 0,C 180,E1 -9260.512,E2 -9260.512} C_VEL
LIN {X 0,Y 440.604,Z 220.969,A -85,B 0,C 180,E1 -9261.87,E2 -9261.87} C_VEL
LIN {X 0,Y 440.489,Z 227.266,A -85,B 0,C 180,E1 -9263.165,E2 -9263.165} C_VEL
LIN {X 0,Y 443.899,Z 244.89,A -85,B 0,C 180,E1 -9263.582,E2 -9263.582} C_VEL
LIN {X 0,Y 443.72,Z 263.293,A -85,B 0,C 180,E1 -9263.88,E2 -9263.88} C_VEL
LIN {X 0,Y 443.006,Z 269.132,A -85,B 0,C 180,E1 -9263.951,E2 -9263.951} C_VEL
LIN {X 0,Y 437.169,Z 288.076,A -85,B 0,C 180,E1 -9264.062,E2 -9264.062} C_VEL
LIN {X 0,Y 436.494,Z 293.913,A -85,B 0,C 180,E1 -9264.136,E2 -9264.136} C_VEL
LIN {X 0,Y 436.032,Z 334.842,A -85,B 0,C 180,E1 -9264.829,E2 -9264.829} C_VEL
LIN {X 0,Y 435.709,Z 347.895,A -85,B 0,C 180,E1 -9265.231,E2 -9265.231} C_VEL
LIN {X 0,Y 435.364,Z 359.881,A -85,B 0,C 180,E1 -9265.778,E2 -9265.778} C_VEL
LIN {X 0,Y 434.924,Z 372.027,A -85,B 0,C 180,E1 -9266.528,E2 -9266.528} C_VEL
LIN {X 0,Y 434.209,Z 383.55,A -85,B 0,C 180,E1 -9267.451,E2 -9267.451} C_VEL
LIN {X 0,Y 433.643,Z 393.889,A -85,B 0,C 180,E1 -9268.493,E2 -9268.493} C_VEL
LIN {X 0,Y 433.107,Z 402.365,A -85,B 0,C 180,E1 -9269.537,E2 -9269.537} C_VEL
LIN {X 0,Y 432.663,Z 410.178,A -85,B 0,C 180,E1 -9270.7,E2 -9270.7} C_VEL
LIN {X 0,Y 432.133,Z 417.845,A -85,B 0,C 180,E1 -9272.099,E2 -9272.099} C_VEL
LIN {X 0,Y 431.84,Z 424.879,A -85,B 0,C 180,E1 -9273.734,E2 -9273.734} C_VEL
LIN {X 0,Y 431.566,Z 429.587,A -85,B 0,C 180,E1 -9275.14,E2 -9275.14} C_VEL
LIN {X 0,Y 431.464,Z 433.186,A -85,B 0,C 180,E1 -9276.548,E2 -9276.548} C_VEL
LIN {X 0,Y 431.343,Z 435.051,A -85,B 0,C 180,E1 -9277.491,E2 -9277.491} C_VEL
LIN {X 0,Y 431.262,Z 436.447,A -85,B 0,C 180,E1 -9278.435,E2 -9278.435} C_VEL
LIN {X 0,Y 431.209,Z 438.048,A -85,B 0,C 180,E1 -9280.329,E2 -9280.329} C_VEL
LIN {X 0,Y 431.258,Z 438.077,A -85,B 0,C 180,E1 -9282.096,E2 -9282.096} C_VEL
LIN {X 0,Y 431.226,Z 437.38,A -85,B 0,C 180,E1 -9283.19,E2 -9283.19} C_VEL
LIN {X 0,Y 431.277,Z 436.351,A -85,B 0,C 180,E1 -9284.149,E2 -9284.149} C_VEL
LIN {X 0,Y 431.408,Z 434.865,A -85,B 0,C 180,E1 -9285.109,E2 -9285.109} C_VEL
LIN {X 0,Y 431.622,Z 431.921,A -85,B 0,C 180,E1 -9286.507,E2 -9286.507} C_VEL
LIN {X 0,Y 431.86,Z 427.604,A -85,B 0,C 180,E1 -9288.011,E2 -9288.011} C_VEL
LIN {X 0,Y 432.27,Z 421.639,A -85,B 0,C 180,E1 -9289.593,E2 -9289.593} C_VEL
LIN {X 0,Y 432.755,Z 415.262,A -85,B 0,C 180,E1 -9290.933,E2 -9290.933} C_VEL
LIN {X 0,Y 433.34,Z 407.985,A -85,B 0,C 180,E1 -9292.182,E2 -9292.182} C_VEL
LIN {X 0,Y 433.99,Z 399.54,A -85,B 0,C 180,E1 -9293.375,E2 -9293.375} C_VEL
LIN {X 0,Y 434.591,Z 389.957,A -85,B 0,C 180,E1 -9294.481,E2 -9294.481} C_VEL
LIN {X 0,Y 435.441,Z 378.147,A -85,B 0,C 180,E1 -9295.561,E2 -9295.561} C_VEL
LIN {X 0,Y 435.976,Z 367.804,A -85,B 0,C 180,E1 -9296.314,E2 -9296.314} C_VEL
LIN {X 0,Y 436.51,Z 355.817,A -85,B 0,C 180,E1 -9296.989,E2 -9296.989} C_VEL
LIN {X 0,Y 436.935,Z 343.651,A -85,B 0,C 180,E1 -9297.479,E2 -9297.479} C_VEL
LIN {X 0,Y 437.195,Z 330.944,A -85,B 0,C 180,E1 -9297.809,E2 -9297.809} C_VEL
LIN {X 0,Y 438.158,Z 244.793,A -85,B 0,C 180,E1 -9299.253,E2 -9299.253} C_VEL
LIN {X 0,Y 434.156,Z 227.622,A -85,B 0,C 180,E1 -9299.769,E2 -9299.769} C_VEL
LIN {X 0,Y 434.118,Z 224.382,A -85,B 0,C 180,E1 -9300.468,E2 -9300.468} C_VEL
LIN {X 0,Y 432.379,Z 215.626,A -85,B 0,C 180,E1 -9302.506,E2 -9302.506} C_VEL
LIN {X 0,Y 432.335,Z 215.633,A -85,B 0,C 180,E1 -9305.816,E2 -9305.816} C_VEL
LIN {X 0,Y 432.358,Z 215.631,A -85,B 0,C 180,E1 -9309.34,E2 -9309.34} C_VEL
LIN {X 0,Y 432.357,Z 215.632,A -85,B 0,C 180,E1 -9311.792,E2 -9311.792} C_VEL
LIN {X 0,Y 432.351,Z 215.629,A -85,B 0,C 180,E1 -9315.659,E2 -9315.659} C_VEL
LIN {X 0,Y 432.359,Z 215.63,A -85,B 0,C 180,E1 -9318.391,E2 -9318.391} C_VEL
LIN {X 0,Y 432.335,Z 215.634,A -85,B 0,C 180,E1 -9321.849,E2 -9321.849} C_VEL
LIN {X 0,Y 432.323,Z 215.631,A -85,B 0,C 180,E1 -9325.321,E2 -9325.321} C_VEL
LIN {X 0,Y 432.303,Z 215.629,A -85,B 0,C 180,E1 -9328.652,E2 -9328.652} C_VEL
LIN {X 0,Y 432.36,Z 215.628,A -85,B 0,C 180,E1 -9331.368,E2 -9331.368} C_VEL
LIN {X 0,Y 432.342,Z 215.632,A -85,B 0,C 180,E1 -9333.966,E2 -9333.966} C_VEL
LIN {X 0,Y 432.296,Z 215.63,A -85,B 0,C 180,E1 -9337.034,E2 -9337.034} C_VEL
LIN {X 0,Y 432.361,Z 215.62,A -85,B 0,C 180,E1 -9340.514,E2 -9340.514} C_VEL
LIN {X 0,Y 432.415,Z 215.616,A -85,B 0,C 180,E1 -9343.96,E2 -9343.96} C_VEL
LIN {X 0,Y 432.431,Z 215.617,A -85,B 0,C 180,E1 -9347.802,E2 -9347.802} C_VEL
LIN {X 0,Y 432.463,Z 215.616,A -85,B 0,C 180,E1 -9351.59,E2 -9351.59} C_VEL
LIN {X 0,Y 432.572,Z 215.595,A -85,B 0,C 180,E1 -9354.406,E2 -9354.406} C_VEL
LIN {X 0,Y 432.571,Z 215.593,A -85,B 0,C 180,E1 -9358.138,E2 -9358.138} C_VEL
LIN {X 0,Y 432.699,Z 215.583,A -85,B 0,C 180,E1 -9360,E2 -9360} C_VEL
LIN {X 0,Y 432.559,Z 215.601,A -85,B 0,C 180,E1 -9362.794,E2 -9362.794} C_VEL
LIN {X 0,Y 432.555,Z 215.602,A -85,B 0,C 180,E1 -9365.594,E2 -9365.594} C_VEL
LIN {X 0,Y 432.435,Z 215.611,A -85,B 0,C 180,E1 -9368.411,E2 -9368.411} C_VEL
LIN {X 0,Y 432.444,Z 215.61,A -85,B 0,C 180,E1 -9372.197,E2 -9372.197} C_VEL
LIN {X 0,Y 432.401,Z 215.618,A -85,B 0,C 180,E1 -9376.04,E2 -9376.04} C_VEL
LIN {X 0,Y 432.36,Z 215.625,A -85,B 0,C 180,E1 -9379.486,E2 -9379.486} C_VEL
LIN {X 0,Y 432.289,Z 215.639,A -85,B 0,C 180,E1 -9382.966,E2 -9382.966} C_VEL
LIN {X 0,Y 432.312,Z 215.629,A -85,B 0,C 180,E1 -9385.004,E2 -9385.004} C_VEL
LIN {X 0,Y 432.321,Z 215.632,A -85,B 0,C 180,E1 -9388.128,E2 -9388.128} C_VEL
LIN {X 0,Y 432.293,Z 215.634,A -85,B 0,C 180,E1 -9391.348,E2 -9391.348} C_VEL
LIN {X 0,Y 432.308,Z 215.636,A -85,B 0,C 180,E1 -9394.68,E2 -9394.68} C_VEL
LIN {X 0,Y 432.315,Z 215.622,A -85,B 0,C 180,E1 -9398.152,E2 -9398.152} C_VEL
LIN {X 0,Y 432.315,Z 215.632,A -85,B 0,C 180,E1 -9401.603,E2 -9401.603} C_VEL
LIN {X 0,Y 432.32,Z 215.635,A -85,B 0,C 180,E1 -9404.349,E2 -9404.349} C_VEL
LIN {X 0,Y 432.305,Z 215.632,A -85,B 0,C 180,E1 -9407.018,E2 -9407.018} C_VEL
LIN {X 0,Y 432.281,Z 215.638,A -85,B 0,C 180,E1 -9409.829,E2 -9409.829} C_VEL
LIN {X 0,Y 432.298,Z 215.635,A -85,B 0,C 180,E1 -9413.023,E2 -9413.023} C_VEL
LIN {X 0,Y 432.354,Z 215.633,A -85,B 0,C 180,E1 -9415.998,E2 -9415.998} C_VEL
LIN {X 0,Y 432.343,Z 215.632,A -85,B 0,C 180,E1 -9419.491,E2 -9419.491} C_VEL
LIN {X 0,Y 432.392,Z 215.706,A -85,B 0,C 180,E1 -9421.944,E2 -9421.944} C_VEL
LIN {X 0,Y 435.234,Z 229.047,A -85,B 0,C 180,E1 -9424.725,E2 -9424.725} C_VEL
LIN {X 0,Y 435.591,Z 232.744,A -85,B 0,C 180,E1 -9425.452,E2 -9425.452} C_VEL
LIN {X 0,Y 434.536,Z 248.753,A -85,B 0,C 180,E1 -9428.411,E2 -9428.411} C_VEL
LIN {X 0,Y 433.738,Z 264.544,A -85,B 0,C 180,E1 -9431.275,E2 -9431.275} C_VEL
LIN {X 0,Y 437.314,Z 286.832,A -85,B 0,C 180,E1 -9431.84,E2 -9431.84} C_VEL
LIN {X 0,Y 437.738,Z 292.322,A -85,B 0,C 180,E1 -9431.954,E2 -9431.954} C_VEL
LIN {X 0,Y 436.904,Z 372.983,A -85,B 0,C 180,E1 -9433.319,E2 -9433.319} C_VEL
LIN {X 0,Y 436.396,Z 386.255,A -85,B 0,C 180,E1 -9433.72,E2 -9433.72} C_VEL
LIN {X 0,Y 435.681,Z 399.539,A -85,B 0,C 180,E1 -9434.324,E2 -9434.324} C_VEL
LIN {X 0,Y 434.988,Z 410.711,A -85,B 0,C 180,E1 -9435.018,E2 -9435.018} C_VEL
LIN {X 0,Y 434.265,Z 422.315,A -85,B 0,C 180,E1 -9435.95,E2 -9435.95} C_VEL
LIN {X 0,Y 433.522,Z 432.777,A -85,B 0,C 180,E1 -9437.001,E2 -9437.001} C_VEL
LIN {X 0,Y 432.972,Z 441.347,A -85,B 0,C 180,E1 -9438.055,E2 -9438.055} C_VEL
LIN {X 0,Y 432.337,Z 449.266,A -85,B 0,C 180,E1 -9439.225,E2 -9439.225} C_VEL
LIN {X 0,Y 431.877,Z 457.034,A -85,B 0,C 180,E1 -9440.634,E2 -9440.634} C_VEL
LIN {X 0,Y 431.532,Z 463.28,A -85,B 0,C 180,E1 -9442.042,E2 -9442.042} C_VEL
LIN {X 0,Y 431.322,Z 468.999,A -85,B 0,C 180,E1 -9443.69,E2 -9443.69} C_VEL
LIN {X 0,Y 431.27,Z 473.199,A -85,B 0,C 180,E1 -9445.325,E2 -9445.325} C_VEL
LIN {X 0,Y 431.192,Z 474.961,A -85,B 0,C 180,E1 -9446.26,E2 -9446.26} C_VEL
LIN {X 0,Y 431.279,Z 476.312,A -85,B 0,C 180,E1 -9447.196,E2 -9447.196} C_VEL
LIN {X 0,Y 431.241,Z 477.263,A -85,B 0,C 180,E1 -9448.131,E2 -9448.131} C_VEL
LIN {X 0,Y 431.222,Z 477.823,A -85,B 0,C 180,E1 -9449.064,E2 -9449.064} C_VEL
LIN {X 0,Y 431.225,Z 477.949,A -85,B 0,C 180,E1 -9449.998,E2 -9449.998} C_VEL
LIN {X 0,Y 431.24,Z 477.019,A -85,B 0,C 180,E1 -9451.866,E2 -9451.866} C_VEL
LIN {X 0,Y 431.297,Z 475.968,A -85,B 0,C 180,E1 -9452.8,E2 -9452.8} C_VEL
LIN {X 0,Y 431.198,Z 474.455,A -85,B 0,C 180,E1 -9453.736,E2 -9453.736} C_VEL
LIN {X 0,Y 431.312,Z 471.398,A -85,B 0,C 180,E1 -9455.139,E2 -9455.139} C_VEL
LIN {X 0,Y 431.374,Z 467.266,A -85,B 0,C 180,E1 -9456.546,E2 -9456.546} C_VEL
LIN {X 0,Y 431.583,Z 460.93,A -85,B 0,C 180,E1 -9458.189,E2 -9458.189} C_VEL
LIN {X 0,Y 431.871,Z 454.025,A -85,B 0,C 180,E1 -9459.599,E2 -9459.599} C_VEL
LIN {X 0,Y 432.231,Z 446.974,A -85,B 0,C 180,E1 -9460.774,E2 -9460.774} C_VEL
LIN {X 0,Y 432.793,Z 438.486,A -85,B 0,C 180,E1 -9461.946,E2 -9461.946} C_VEL
LIN {X 0,Y 433.368,Z 427.98,A -85,B 0,C 180,E1 -9463.12,E2 -9463.12} C_VEL
LIN {X 0,Y 434.04,Z 416.14,A -85,B 0,C 180,E1 -9464.173,E2 -9464.173} C_VEL
LIN {X 0,Y 434.676,Z 404.273,A -85,B 0,C 180,E1 -9464.989,E2 -9464.989} C_VEL
LIN {X 0,Y 435.277,Z 391.924,A -85,B 0,C 180,E1 -9465.627,E2 -9465.627} C_VEL
LIN {X 0,Y 435.775,Z 379.293,A -85,B 0,C 180,E1 -9466.089,E2 -9466.089} C_VEL
LIN {X 0,Y 436.079,Z 366.277,A -85,B 0,C 180,E1 -9466.378,E2 -9466.378} C_VEL
LIN {X 0,Y 436.666,Z 289.095,A -85,B 0,C 180,E1 -9467.65,E2 -9467.65} C_VEL
LIN {X 0,Y 433.247,Z 264.75,A -85,B 0,C 180,E1 -9468.192,E2 -9468.192} C_VEL
LIN {X 0,Y 434.174,Z 245.686,A -85,B 0,C 180,E1 -9471.604,E2 -9471.604} C_VEL
LIN {X 0,Y 434.96,Z 229.247,A -85,B 0,C 180,E1 -9474.582,E2 -9474.582} C_VEL
LIN {X 0,Y 432.642,Z 216.572,A -85,B 0,C 180,E1 -9477.05,E2 -9477.05} C_VEL
LIN {X 0,Y 432.454,Z 215.618,A -85,B 0,C 180,E1 -9477.259,E2 -9477.259} C_VEL
LIN {X 0,Y 432.331,Z 215.63,A -85,B 0,C 180,E1 -9480.506,E2 -9480.506} C_VEL
LIN {X 0,Y 432.34,Z 215.634,A -85,B 0,C 180,E1 -9483.999,E2 -9483.999} C_VEL
LIN {X 0,Y 432.3,Z 215.632,A -85,B 0,C 180,E1 -9487.193,E2 -9487.193} C_VEL
LIN {X 0,Y 432.307,Z 215.635,A -85,B 0,C 180,E1 -9490.175,E2 -9490.175} C_VEL
LIN {X 0,Y 432.289,Z 215.633,A -85,B 0,C 180,E1 -9493.057,E2 -9493.057} C_VEL
LIN {X 0,Y 432.331,Z 215.633,A -85,B 0,C 180,E1 -9495.657,E2 -9495.657} C_VEL
LIN {X 0,Y 432.34,Z 215.628,A -85,B 0,C 180,E1 -9498.388,E2 -9498.388} C_VEL
LIN {X 0,Y 432.317,Z 215.635,A -85,B 0,C 180,E1 -9501.848,E2 -9501.848} C_VEL
LIN {X 0,Y 432.301,Z 215.635,A -85,B 0,C 180,E1 -9505.319,E2 -9505.319} C_VEL
LIN {X 0,Y 432.281,Z 215.634,A -85,B 0,C 180,E1 -9508.651,E2 -9508.651} C_VEL
LIN {X 0,Y 432.337,Z 215.632,A -85,B 0,C 180,E1 -9511.366,E2 -9511.366} C_VEL
LIN {X 0,Y 432.322,Z 215.631,A -85,B 0,C 180,E1 -9513.965,E2 -9513.965} C_VEL
LIN {X 0,Y 432.287,Z 215.636,A -85,B 0,C 180,E1 -9517.034,E2 -9517.034} C_VEL
LIN {X 0,Y 432.339,Z 215.628,A -85,B 0,C 180,E1 -9520.04,E2 -9520.04} C_VEL
LIN {X 0,Y 432.371,Z 215.628,A -85,B 0,C 180,E1 -9523.515,E2 -9523.515} C_VEL
LIN {X 0,Y 432.393,Z 215.627,A -85,B 0,C 180,E1 -9527.187,E2 -9527.187} C_VEL
LIN {X 0,Y 432.402,Z 215.62,A -85,B 0,C 180,E1 -9530.646,E2 -9530.646} C_VEL
LIN {X 0,Y 432.55,Z 215.604,A -85,B 0,C 180,E1 -9533.469,E2 -9533.469} C_VEL
LIN {X 0,Y 432.556,Z 215.606,A -85,B 0,C 180,E1 -9537.206,E2 -9537.206} C_VEL
LIN {X 0,Y 432.675,Z 215.585,A -85,B 0,C 180,E1 -9540,E2 -9540} C_VEL
LIN {X 0,Y 432.536,Z 215.607,A -85,B 0,C 180,E1 -9542.794,E2 -9542.794} C_VEL
LIN {X 0,Y 432.513,Z 215.608,A -85,B 0,C 180,E1 -9546.531,E2 -9546.531} C_VEL
LIN {X 0,Y 432.391,Z 215.622,A -85,B 0,C 180,E1 -9549.354,E2 -9549.354} C_VEL
LIN {X 0,Y 432.393,Z 215.628,A -85,B 0,C 180,E1 -9552.813,E2 -9552.813} C_VEL
LIN {X 0,Y 432.371,Z 215.627,A -85,B 0,C 180,E1 -9556.485,E2 -9556.485} C_VEL
LIN {X 0,Y 432.288,Z 215.634,A -85,B 0,C 180,E1 -9559.963,E2 -9559.963} C_VEL
LIN {X 0,Y 432.271,Z 215.639,A -85,B 0,C 180,E1 -9562.967,E2 -9562.967} C_VEL
LIN {X 0,Y 432.318,Z 215.631,A -85,B 0,C 180,E1 -9566.036,E2 -9566.036} C_VEL
LIN {X 0,Y 432.309,Z 215.631,A -85,B 0,C 180,E1 -9569.19,E2 -9569.19} C_VEL
LIN {X 0,Y 432.284,Z 215.639,A -85,B 0,C 180,E1 -9572.297,E2 -9572.297} C_VEL
LIN {X 0,Y 432.301,Z 215.636,A -85,B 0,C 180,E1 -9574.681,E2 -9574.681} C_VEL
LIN {X 0,Y 432.305,Z 215.636,A -85,B 0,C 180,E1 -9578.154,E2 -9578.154} C_VEL
LIN {X 0,Y 432.337,Z 215.628,A -85,B 0,C 180,E1 -9581.612,E2 -9581.612} C_VEL
LIN {X 0,Y 432.332,Z 215.634,A -85,B 0,C 180,E1 -9584.348,E2 -9584.348} C_VEL
LIN {X 0,Y 432.293,Z 215.633,A -85,B 0,C 180,E1 -9587.02,E2 -9587.02} C_VEL
LIN {X 0,Y 432.316,Z 215.633,A -85,B 0,C 180,E1 -9589.824,E2 -9589.824} C_VEL
LIN {X 0,Y 432.285,Z 215.633,A -85,B 0,C 180,E1 -9593.026,E2 -9593.026} C_VEL
LIN {X 0,Y 432.341,Z 215.633,A -85,B 0,C 180,E1 -9596.001,E2 -9596.001} C_VEL
LIN {X 0,Y 432.332,Z 215.63,A -85,B 0,C 180,E1 -9599.494,E2 -9599.494} C_VEL
LIN {X 0,Y 432.378,Z 215.622,A -85,B 0,C 180,E1 -9602.932,E2 -9602.932} C_VEL
LIN {X 0,Y 432.358,Z 215.63,A -85,B 0,C 180,E1 -9606.027,E2 -9606.027} C_VEL
LIN {X 0,Y 432.342,Z 215.627,A -85,B 0,C 180,E1 -9609.05,E2 -9609.05} C_VEL
LIN {X 0,Y 432.354,Z 215.629,A -85,B 0,C 180,E1 -9612.014,E2 -9612.014} C_VEL
LIN {X 0,Y 432.39,Z 215.621,A -85,B 0,C 180,E1 -9614.93,E2 -9614.93} C_VEL
LIN {X 0,Y 432.458,Z 215.619,A -85,B 0,C 180,E1 -9617.806,E2 -9617.806} C_VEL
LIN {X 0,Y 432.489,Z 215.74,A -85,B 0,C 180,E1 -9620.356,E2 -9620.356} C_VEL
LIN {X 0,Y 433.7,Z 223.546,A -85,B 0,C 180,E1 -9622.085,E2 -9622.085} C_VEL
LIN {X 0,Y 433.549,Z 227.425,A -85,B 0,C 180,E1 -9622.902,E2 -9622.902} C_VEL
LIN {X 0,Y 437.024,Z 245.128,A -85,B 0,C 180,E1 -9623.336,E2 -9623.336} C_VEL
LIN {X 0,Y 436.494,Z 293.913,A -85,B 0,C 180,E1 -9624.136,E2 -9624.136} C_VEL
LIN {X 0,Y 435.814,Z 299.756,A -85,B 0,C 180,E1 -9624.21,E2 -9624.21} C_VEL
LIN {X 0,Y 429.995,Z 318.717,A -85,B 0,C 180,E1 -9624.328,E2 -9624.328} C_VEL
LIN {X 0,Y 429.327,Z 324.559,A -85,B 0,C 180,E1 -9624.405,E2 -9624.405} C_VEL
LIN {X 0,Y 429.128,Z 338.338,A -85,B 0,C 180,E1 -9624.687,E2 -9624.687} C_VEL
LIN {X 0,Y 428.823,Z 351.036,A -85,B 0,C 180,E1 -9625.125,E2 -9625.125} C_VEL
LIN {X 0,Y 428.293,Z 363.75,A -85,B 0,C 180,E1 -9625.767,E2 -9625.767} C_VEL
LIN {X 0,Y 427.788,Z 375.832,A -85,B 0,C 180,E1 -9626.588,E2 -9626.588} C_VEL
LIN {X 0,Y 427.104,Z 386.672,A -85,B 0,C 180,E1 -9627.526,E2 -9627.526} C_VEL
LIN {X 0,Y 426.542,Z 396.444,A -85,B 0,C 180,E1 -9628.586,E2 -9628.586} C_VEL
LIN {X 0,Y 425.966,Z 405.349,A -85,B 0,C 180,E1 -9629.765,E2 -9629.765} C_VEL
LIN {X 0,Y 425.385,Z 414.058,A -85,B 0,C 180,E1 -9631.185,E2 -9631.185} C_VEL
LIN {X 0,Y 424.937,Z 421.025,A -85,B 0,C 180,E1 -9632.608,E2 -9632.608} C_VEL
LIN {X 0,Y 424.671,Z 427.392,A -85,B 0,C 180,E1 -9634.272,E2 -9634.272} C_VEL
LIN {X 0,Y 424.47,Z 431.602,A -85,B 0,C 180,E1 -9635.703,E2 -9635.703} C_VEL
LIN {X 0,Y 424.354,Z 433.843,A -85,B 0,C 180,E1 -9636.658,E2 -9636.658} C_VEL
LIN {X 0,Y 424.255,Z 435.609,A -85,B 0,C 180,E1 -9637.617,E2 -9637.617} C_VEL
LIN {X 0,Y 424.157,Z 436.95,A -85,B 0,C 180,E1 -9638.577,E2 -9638.577} C_VEL
LIN {X 0,Y 424.116,Z 438.444,A -85,B 0,C 180,E1 -9640.503,E2 -9640.503} C_VEL
LIN {X 0,Y 424.165,Z 438.403,A -85,B 0,C 180,E1 -9642.156,E2 -9642.156} C_VEL
LIN {X 0,Y 424.15,Z 437.585,A -85,B 0,C 180,E1 -9643.414,E2 -9643.414} C_VEL
LIN {X 0,Y 424.214,Z 436.482,A -85,B 0,C 180,E1 -9644.39,E2 -9644.39} C_VEL
LIN {X 0,Y 424.503,Z 433.217,A -85,B 0,C 180,E1 -9646.21,E2 -9646.21} C_VEL
LIN {X 0,Y 424.778,Z 429.003,A -85,B 0,C 180,E1 -9647.823,E2 -9647.823} C_VEL
LIN {X 0,Y 425.147,Z 423.881,A -85,B 0,C 180,E1 -9649.306,E2 -9649.306} C_VEL
LIN {X 0,Y 425.686,Z 417.349,A -85,B 0,C 180,E1 -9650.791,E2 -9650.791} C_VEL
LIN {X 0,Y 426.365,Z 409.093,A -85,B 0,C 180,E1 -9652.279,E2 -9652.279} C_VEL
LIN {X 0,Y 427.049,Z 400.59,A -85,B 0,C 180,E1 -9653.52,E2 -9653.52} C_VEL
LIN {X 0,Y 427.691,Z 391.22,A -85,B 0,C 180,E1 -9654.643,E2 -9654.643} C_VEL
LIN {X 0,Y 428.529,Z 380.473,A -85,B 0,C 180,E1 -9655.67,E2 -9655.67} C_VEL
LIN {X 0,Y 429.164,Z 369.592,A -85,B 0,C 180,E1 -9656.502,E2 -9656.502} C_VEL
LIN {X 0,Y 429.691,Z 358.071,A -85,B 0,C 180,E1 -9657.189,E2 -9657.189} C_VEL
LIN {X 0,Y 430.189,Z 345.598,A -85,B 0,C 180,E1 -9657.731,E2 -9657.731} C_VEL
LIN {X 0,Y 430.465,Z 333.365,A -85,B 0,C 180,E1 -9658.079,E2 -9658.079} C_VEL
LIN {X 0,Y 431.606,Z 246.156,A -85,B 0,C 180,E1 -9659.564,E2 -9659.564} C_VEL
LIN {X 0,Y 427.281,Z 228.008,A -85,B 0,C 180,E1 -9660.116,E2 -9660.116} C_VEL
LIN {X 0,Y 426.591,Z 222.383,A -85,B 0,C 180,E1 -9661.393,E2 -9661.393} C_VEL
LIN {X 0,Y 425.322,Z 216.504,A -85,B 0,C 180,E1 -9662.834,E2 -9662.834} C_VEL
LIN {X 0,Y 425.28,Z 216.512,A -85,B 0,C 180,E1 -9665.928,E2 -9665.928} C_VEL
LIN {X 0,Y 425.303,Z 216.51,A -85,B 0,C 180,E1 -9669.044,E2 -9669.044} C_VEL
LIN {X 0,Y 425.306,Z 216.512,A -85,B 0,C 180,E1 -9671.96,E2 -9671.96} C_VEL
LIN {X 0,Y 425.292,Z 216.507,A -85,B 0,C 180,E1 -9675.279,E2 -9675.279} C_VEL
LIN {X 0,Y 425.295,Z 216.508,A -85,B 0,C 180,E1 -9678.623,E2 -9678.623} C_VEL
LIN {X 0,Y 425.306,Z 216.505,A -85,B 0,C 180,E1 -9681.102,E2 -9681.102} C_VEL
LIN {X 0,Y 425.283,Z 216.507,A -85,B 0,C 180,E1 -9684.662,E2 -9684.662} C_VEL
LIN {X 0,Y 425.247,Z 216.513,A -85,B 0,C 180,E1 -9688.071,E2 -9688.071} C_VEL
LIN {X 0,Y 425.317,Z 216.505,A -85,B 0,C 180,E1 -9691.367,E2 -9691.367} C_VEL
LIN {X 0,Y 425.273,Z 216.508,A -85,B 0,C 180,E1 -9694.553,E2 -9694.553} C_VEL
LIN {X 0,Y 425.265,Z 216.512,A -85,B 0,C 180,E1 -9697.66,E2 -9697.66} C_VEL
LIN {X 0,Y 425.336,Z 216.495,A -85,B 0,C 180,E1 -9700.703,E2 -9700.703} C_VEL
LIN {X 0,Y 425.372,Z 216.496,A -85,B 0,C 180,E1 -9703.687,E2 -9703.687} C_VEL
LIN {X 0,Y 425.384,Z 216.497,A -85,B 0,C 180,E1 -9707.597,E2 -9707.597} C_VEL
LIN {X 0,Y 425.414,Z 216.496,A -85,B 0,C 180,E1 -9711.449,E2 -9711.449} C_VEL
LIN {X 0,Y 425.529,Z 216.473,A -85,B 0,C 180,E1 -9714.313,E2 -9714.313} C_VEL
LIN {X 0,Y 425.54,Z 216.469,A -85,B 0,C 180,E1 -9718.107,E2 -9718.107} C_VEL
LIN {X 0,Y 425.669,Z 216.458,A -85,B 0,C 180,E1 -9720,E2 -9720} C_VEL
LIN {X 0,Y 425.513,Z 216.478,A -85,B 0,C 180,E1 -9722.84,E2 -9722.84} C_VEL
LIN {X 0,Y 425.511,Z 216.478,A -85,B 0,C 180,E1 -9725.687,E2 -9725.687} C_VEL
LIN {X 0,Y 425.38,Z 216.491,A -85,B 0,C 180,E1 -9728.551,E2 -9728.551} C_VEL
LIN {X 0,Y 425.394,Z 216.49,A -85,B 0,C 180,E1 -9732.402,E2 -9732.402} C_VEL
LIN {X 0,Y 425.36,Z 216.497,A -85,B 0,C 180,E1 -9736.313,E2 -9736.313} C_VEL
LIN {X 0,Y 425.302,Z 216.504,A -85,B 0,C 180,E1 -9739.636,E2 -9739.636} C_VEL
LIN {X 0,Y 425.263,Z 216.507,A -85,B 0,C 180,E1 -9742.34,E2 -9742.34} C_VEL
LIN {X 0,Y 425.294,Z 216.508,A -85,B 0,C 180,E1 -9744.658,E2 -9744.658} C_VEL
LIN {X 0,Y 425.247,Z 216.512,A -85,B 0,C 180,E1 -9747.565,E2 -9747.565} C_VEL
LIN {X 0,Y 425.268,Z 216.513,A -85,B 0,C 180,E1 -9750.762,E2 -9750.762} C_VEL
LIN {X 0,Y 425.272,Z 216.508,A -85,B 0,C 180,E1 -9754.285,E2 -9754.285} C_VEL
LIN {X 0,Y 425.26,Z 216.503,A -85,B 0,C 180,E1 -9757.696,E2 -9757.696} C_VEL
LIN {X 0,Y 425.253,Z 216.513,A -85,B 0,C 180,E1 -9760.52,E2 -9760.52} C_VEL
LIN {X 0,Y 425.243,Z 216.512,A -85,B 0,C 180,E1 -9763.352,E2 -9763.352} C_VEL
LIN {X 0,Y 425.244,Z 216.514,A -85,B 0,C 180,E1 -9766.651,E2 -9766.651} C_VEL
LIN {X 0,Y 425.235,Z 216.516,A -85,B 0,C 180,E1 -9769.869,E2 -9769.869} C_VEL
LIN {X 0,Y 425.269,Z 216.512,A -85,B 0,C 180,E1 -9772.49,E2 -9772.49} C_VEL
LIN {X 0,Y 425.302,Z 216.51,A -85,B 0,C 180,E1 -9775.818,E2 -9775.818} C_VEL
LIN {X 0,Y 425.287,Z 216.511,A -85,B 0,C 180,E1 -9779.24,E2 -9779.24} C_VEL
LIN {X 0,Y 425.339,Z 216.658,A -85,B 0,C 180,E1 -9781.639,E2 -9781.639} C_VEL
LIN {X 0,Y 428.254,Z 230.097,A -85,B 0,C 180,E1 -9784.502,E2 -9784.502} C_VEL
LIN {X 0,Y 428.726,Z 234.009,A -85,B 0,C 180,E1 -9785.291,E2 -9785.291} C_VEL
LIN {X 0,Y 427.607,Z 250.005,A -85,B 0,C 180,E1 -9788.297,E2 -9788.297} C_VEL
LIN {X 0,Y 426.8,Z 264.073,A -85,B 0,C 180,E1 -9790.91,E2 -9790.91} C_VEL
LIN {X 0,Y 430.589,Z 286.827,A -85,B 0,C 180,E1 -9791.507,E2 -9791.507} C_VEL
LIN {X 0,Y 431.107,Z 292.352,A -85,B 0,C 180,E1 -9791.63,E2 -9791.63} C_VEL
LIN {X 0,Y 430.195,Z 373.062,A -85,B 0,C 180,E1 -9793.021,E2 -9793.021} C_VEL
LIN {X 0,Y 429.613,Z 386.948,A -85,B 0,C 180,E1 -9793.456,E2 -9793.456} C_VEL
LIN {X 0,Y 428.881,Z 399.92,A -85,B 0,C 180,E1 -9794.069,E2 -9794.069} C_VEL
LIN {X 0,Y 428.041,Z 412.487,A -85,B 0,C 180,E1 -9794.891,E2 -9794.891} C_VEL
LIN {X 0,Y 427.289,Z 423.545,A -85,B 0,C 180,E1 -9795.823,E2 -9795.823} C_VEL
LIN {X 0,Y 426.525,Z 433.83,A -85,B 0,C 180,E1 -9796.905,E2 -9796.905} C_VEL
LIN {X 0,Y 425.894,Z 442.977,A -85,B 0,C 180,E1 -9798.095,E2 -9798.095} C_VEL
LIN {X 0,Y 425.122,Z 451.909,A -85,B 0,C 180,E1 -9799.522,E2 -9799.522} C_VEL
LIN {X 0,Y 424.702,Z 459.121,A -85,B 0,C 180,E1 -9800.954,E2 -9800.954} C_VEL
LIN {X 0,Y 424.377,Z 464.897,A -85,B 0,C 180,E1 -9802.386,E2 -9802.386} C_VEL
LIN {X 0,Y 424.217,Z 469.221,A -85,B 0,C 180,E1 -9803.732,E2 -9803.732} C_VEL
LIN {X 0,Y 424.198,Z 472.945,A -85,B 0,C 180,E1 -9805.247,E2 -9805.247} C_VEL
LIN {X 0,Y 424.174,Z 476.024,A -85,B 0,C 180,E1 -9807.149,E2 -9807.149} C_VEL
LIN {X 0,Y 424.165,Z 476.965,A -85,B 0,C 180,E1 -9808.099,E2 -9808.099} C_VEL
LIN {X 0,Y 424.138,Z 477.507,A -85,B 0,C 180,E1 -9809.049,E2 -9809.049} C_VEL
LIN {X 0,Y 424.139,Z 477.616,A -85,B 0,C 180,E1 -9809.998,E2 -9809.998} C_VEL
LIN {X 0,Y 424.165,Z 476.663,A -85,B 0,C 180,E1 -9811.897,E2 -9811.897} C_VEL
LIN {X 0,Y 424.206,Z 475.596,A -85,B 0,C 180,E1 -9812.847,E2 -9812.847} C_VEL
LIN {X 0,Y 424.108,Z 474.061,A -85,B 0,C 180,E1 -9813.798,E2 -9813.798} C_VEL
LIN {X 0,Y 424.22,Z 470.978,A -85,B 0,C 180,E1 -9815.226,E2 -9815.226} C_VEL
LIN {X 0,Y 424.297,Z 466.817,A -85,B 0,C 180,E1 -9816.656,E2 -9816.656} C_VEL
LIN {X 0,Y 424.509,Z 460.447,A -85,B 0,C 180,E1 -9818.327,E2 -9818.327} C_VEL
LIN {X 0,Y 424.838,Z 453.506,A -85,B 0,C 180,E1 -9819.76,E2 -9819.76} C_VEL
LIN {X 0,Y 425.223,Z 446.413,A -85,B 0,C 180,E1 -9820.954,E2 -9820.954} C_VEL
LIN {X 0,Y 425.774,Z 437.86,A -85,B 0,C 180,E1 -9822.146,E2 -9822.146} C_VEL
LIN {X 0,Y 426.412,Z 427.274,A -85,B 0,C 180,E1 -9823.338,E2 -9823.338} C_VEL
LIN {X 0,Y 427.104,Z 415.345,A -85,B 0,C 180,E1 -9824.408,E2 -9824.408} C_VEL
LIN {X 0,Y 427.801,Z 403.301,A -85,B 0,C 180,E1 -9825.236,E2 -9825.236} C_VEL
LIN {X 0,Y 428.442,Z 390.751,A -85,B 0,C 180,E1 -9825.883,E2 -9825.883} C_VEL
LIN {X 0,Y 428.9,Z 378.683,A -85,B 0,C 180,E1 -9826.324,E2 -9826.324} C_VEL
LIN {X 0,Y 429.184,Z 365.375,A -85,B 0,C 180,E1 -9826.618,E2 -9826.618} C_VEL
LIN {X 0,Y 429.78,Z 289.645,A -85,B 0,C 180,E1 -9827.886,E2 -9827.886} C_VEL
LIN {X 0,Y 426.272,Z 264.481,A -85,B 0,C 180,E1 -9828.446,E2 -9828.446} C_VEL
LIN {X 0,Y 427.272,Z 245.112,A -85,B 0,C 180,E1 -9831.971,E2 -9831.971} C_VEL
LIN {X 0,Y 428.004,Z 231.407,A -85,B 0,C 180,E1 -9834.491,E2 -9834.491} C_VEL
LIN {X 0,Y 426.959,Z 224.395,A -85,B 0,C 180,E1 -9835.857,E2 -9835.857} C_VEL
LIN {X 0,Y 425.397,Z 216.498,A -85,B 0,C 180,E1 -9837.464,E2 -9837.464} C_VEL
LIN {X 0,Y 425.271,Z 216.508,A -85,B 0,C 180,E1 -9840.812,E2 -9840.812} C_VEL
LIN {X 0,Y 425.292,Z 216.509,A -85,B 0,C 180,E1 -9844.284,E2 -9844.284} C_VEL
LIN {X 0,Y 425.256,Z 216.513,A -85,B 0,C 180,E1 -9847.69,E2 -9847.69} C_VEL
LIN {X 0,Y 425.253,Z 216.511,A -85,B 0,C 180,E1 -9850.516,E2 -9850.516} C_VEL
LIN {X 0,Y 425.229,Z 216.514,A -85,B 0,C 180,E1 -9853.347,E2 -9853.347} C_VEL
LIN {X 0,Y 425.282,Z 216.506,A -85,B 0,C 180,E1 -9856.637,E2 -9856.637} C_VEL
LIN {X 0,Y 425.278,Z 216.512,A -85,B 0,C 180,E1 -9859.872,E2 -9859.872} C_VEL
LIN {X 0,Y 425.25,Z 216.51,A -85,B 0,C 180,E1 -9862.483,E2 -9862.483} C_VEL
LIN {X 0,Y 425.268,Z 216.513,A -85,B 0,C 180,E1 -9865.814,E2 -9865.814} C_VEL
LIN {X 0,Y 425.257,Z 216.512,A -85,B 0,C 180,E1 -9869.234,E2 -9869.234} C_VEL
LIN {X 0,Y 425.305,Z 216.503,A -85,B 0,C 180,E1 -9872.439,E2 -9872.439} C_VEL
LIN {X 0,Y 425.31,Z 216.508,A -85,B 0,C 180,E1 -9875.6,E2 -9875.6} C_VEL
LIN {X 0,Y 425.286,Z 216.506,A -85,B 0,C 180,E1 -9878.681,E2 -9878.681} C_VEL
LIN {X 0,Y 425.283,Z 216.509,A -85,B 0,C 180,E1 -9881.701,E2 -9881.701} C_VEL
LIN {X 0,Y 425.305,Z 216.504,A -85,B 0,C 180,E1 -9884.669,E2 -9884.669} C_VEL
LIN {X 0,Y 425.379,Z 216.497,A -85,B 0,C 180,E1 -9887.597,E2 -9887.597} C_VEL
LIN {X 0,Y 425.413,Z 216.494,A -85,B 0,C 180,E1 -9891.449,E2 -9891.449} C_VEL
LIN {X 0,Y 425.528,Z 216.475,A -85,B 0,C 180,E1 -9894.313,E2 -9894.313} C_VEL
LIN {X 0,Y 425.519,Z 216.476,A -85,B 0,C 180,E1 -9898.107,E2 -9898.107} C_VEL
LIN {X 0,Y 425.646,Z 216.461,A -85,B 0,C 180,E1 -9900,E2 -9900} C_VEL
LIN {X 0,Y 425.49,Z 216.485,A -85,B 0,C 180,E1 -9902.84,E2 -9902.84} C_VEL
LIN {X 0,Y 425.471,Z 216.486,A -85,B 0,C 180,E1 -9906.64,E2 -9906.64} C_VEL
LIN {X 0,Y 425.35,Z 216.498,A -85,B 0,C 180,E1 -9909.511,E2 -9909.511} C_VEL
LIN {X 0,Y 425.352,Z 216.503,A -85,B 0,C 180,E1 -9912.912,E2 -9912.912} C_VEL
LIN {X 0,Y 425.319,Z 216.507,A -85,B 0,C 180,E1 -9916.61,E2 -9916.61} C_VEL
LIN {X 0,Y 425.278,Z 216.506,A -85,B 0,C 180,E1 -9919.638,E2 -9919.638} C_VEL
LIN {X 0,Y 425.241,Z 216.515,A -85,B 0,C 180,E1 -9922.342,E2 -9922.342} C_VEL
LIN {X 0,Y 425.249,Z 216.51,A -85,B 0,C 180,E1 -9925.449,E2 -9925.449} C_VEL
LIN {X 0,Y 425.294,Z 216.511,A -85,B 0,C 180,E1 -9928.635,E2 -9928.635} C_VEL
LIN {X 0,Y 425.224,Z 216.515,A -85,B 0,C 180,E1 -9931.931,E2 -9931.931} C_VEL
LIN {X 0,Y 425.261,Z 216.508,A -85,B 0,C 180,E1 -9935.34,E2 -9935.34} C_VEL
LIN {X 0,Y 425.271,Z 216.508,A -85,B 0,C 180,E1 -9939.049,E2 -9939.049} C_VEL
LIN {X 0,Y 425.299,Z 216.507,A -85,B 0,C 180,E1 -9942.65,E2 -9942.65} C_VEL
LIN {X 0,Y 425.234,Z 216.517,A -85,B 0,C 180,E1 -9946.048,E2 -9946.048} C_VEL
LIN {X 0,Y 425.249,Z 216.512,A -85,B 0,C 180,E1 -9948.626,E2 -9948.626} C_VEL
LIN {X 0,Y 425.289,Z 216.505,A -85,B 0,C 180,E1 -9951.107,E2 -9951.107} C_VEL
LIN {X 0,Y 425.28,Z 216.507,A -85,B 0,C 180,E1 -9954.668,E2 -9954.668} C_VEL
LIN {X 0,Y 425.249,Z 216.517,A -85,B 0,C 180,E1 -9958.077,E2 -9958.077} C_VEL
LIN {X 0,Y 425.317,Z 216.503,A -85,B 0,C 180,E1 -9961.372,E2 -9961.372} C_VEL
LIN {X 0,Y 425.342,Z 216.501,A -85,B 0,C 180,E1 -9963.509,E2 -9963.509} C_VEL
LIN {X 0,Y 425.276,Z 216.507,A -85,B 0,C 180,E1 -9966.637,E2 -9966.637} C_VEL
LIN {X 0,Y 425.288,Z 216.511,A -85,B 0,C 180,E1 -9969.698,E2 -9969.698} C_VEL
LIN {X 0,Y 425.328,Z 216.5,A -85,B 0,C 180,E1 -9972.7,E2 -9972.7} C_VEL
LIN {X 0,Y 425.343,Z 216.505,A -85,B 0,C 180,E1 -9975.653,E2 -9975.653} C_VEL
LIN {X 0,Y 425.349,Z 216.502,A -85,B 0,C 180,E1 -9978.567,E2 -9978.567} C_VEL
LIN {X 0,Y 425.451,Z 216.676,A -85,B 0,C 180,E1 -9980.195,E2 -9980.195} C_VEL
LIN {X 0,Y 426.736,Z 224.503,A -85,B 0,C 180,E1 -9981.955,E2 -9981.955} C_VEL
LIN {X 0,Y 426.629,Z 227.704,A -85,B 0,C 180,E1 -9982.638,E2 -9982.638} C_VEL
LIN {X 0,Y 430.203,Z 246.908,A -85,B 0,C 180,E1 -9983.112,E2 -9983.112} C_VEL
LIN {X 0,Y 429.327,Z 324.559,A -85,B 0,C 180,E1 -9984.405,E2 -9984.405} C_VEL
LIN {X 0,Y 428.623,Z 330.39,A -85,B 0,C 180,E1 -9984.483,E2 -9984.483} C_VEL
LIN {X 0,Y 425.636,Z 339.805,A -85,B 0,C 180,E1 -9984.606,E2 -9984.606} C_VEL
LIN {X 0,Y 422.647,Z 349.136,A -85,B 0,C 180,E1 -9984.834,E2 -9984.834} C_VEL
LIN {X 0,Y 421.84,Z 354.693,A -85,B 0,C 180,E1 -9985.056,E2 -9985.056} C_VEL
LIN {X 0,Y 421.339,Z 366.411,A -85,B 0,C 180,E1 -9985.698,E2 -9985.698} C_VEL
LIN {X 0,Y 420.741,Z 377.952,A -85,B 0,C 180,E1 -9986.531,E2 -9986.531} C_VEL
LIN {X 0,Y 420.07,Z 388.394,A -85,B 0,C 180,E1 -9987.485,E2 -9987.485} C_VEL
LIN {X 0,Y 419.499,Z 397.933,A -85,B 0,C 180,E1 -9988.562,E2 -9988.562} C_VEL
LIN {X 0,Y 418.906,Z 406.649,A -85,B 0,C 180,E1 -9989.762,E2 -9989.762} C_VEL
LIN {X 0,Y 418.297,Z 415.15,A -85,B 0,C 180,E1 -9991.205,E2 -9991.205} C_VEL
LIN {X 0,Y 417.844,Z 421.958,A -85,B 0,C 180,E1 -9992.653,E2 -9992.653} C_VEL
LIN {X 0,Y 417.565,Z 428.207,A -85,B 0,C 180,E1 -9994.345,E2 -9994.345} C_VEL
LIN {X 0,Y 417.376,Z 432.306,A -85,B 0,C 180,E1 -9995.8,E2 -9995.8} C_VEL
LIN {X 0,Y 417.248,Z 434.466,A -85,B 0,C 180,E1 -9996.772,E2 -9996.772} C_VEL
LIN {X 0,Y 417.143,Z 436.158,A -85,B 0,C 180,E1 -9997.747,E2 -9997.747} C_VEL
LIN {X 0,Y 417.068,Z 437.449,A -85,B 0,C 180,E1 -9998.724,E2 -9998.724} C_VEL
LIN {X 0,Y 417,Z 438.347,A -85,B 0,C 180,E1 -9999.704,E2 -9999.704} C_VEL
LIN {X 0,Y 417.035,Z 438.803,A -85,B 0,C 180,E1 -10000.684,E2 -10000.684} C_VEL
LIN {X 0,Y 417.079,Z 438.728,A -85,B 0,C 180,E1 -10002.222,E2 -10002.222} C_VEL
LIN {X 0,Y 417.071,Z 437.786,A -85,B 0,C 180,E1 -10003.646,E2 -10003.646} C_VEL
LIN {X 0,Y 417.157,Z 436.588,A -85,B 0,C 180,E1 -10004.638,E2 -10004.638} C_VEL
LIN {X 0,Y 417.453,Z 433.551,A -85,B 0,C 180,E1 -10006.337,E2 -10006.337} C_VEL
LIN {X 0,Y 417.787,Z 428.889,A -85,B 0,C 180,E1 -10008.132,E2 -10008.132} C_VEL
LIN {X 0,Y 418.246,Z 423.048,A -85,B 0,C 180,E1 -10009.779,E2 -10009.779} C_VEL
LIN {X 0,Y 418.902,Z 415.649,A -85,B 0,C 180,E1 -10011.401,E2 -10011.401} C_VEL
LIN {X 0,Y 419.535,Z 408.502,A -85,B 0,C 180,E1 -10012.662,E2 -10012.662} C_VEL
LIN {X 0,Y 420.306,Z 398.788,A -85,B 0,C 180,E1 -10014.052,E2 -10014.052} C_VEL
LIN {X 0,Y 421.095,Z 388.904,A -85,B 0,C 180,E1 -10015.187,E2 -10015.187} C_VEL
LIN {X 0,Y 421.903,Z 378.607,A -85,B 0,C 180,E1 -10016.141,E2 -10016.141} C_VEL
LIN {X 0,Y 422.574,Z 366.735,A -85,B 0,C 180,E1 -10017.016,E2 -10017.016} C_VEL
LIN {X 0,Y 423.139,Z 355.411,A -85,B 0,C 180,E1 -10017.646,E2 -10017.646} C_VEL
LIN {X 0,Y 423.611,Z 342.282,A -85,B 0,C 180,E1 -10018.169,E2 -10018.169} C_VEL
LIN {X 0,Y 423.898,Z 329.465,A -85,B 0,C 180,E1 -10018.484,E2 -10018.484} C_VEL
LIN {X 0,Y 424.903,Z 246.725,A -85,B 0,C 180,E1 -10019.91,E2 -10019.91} C_VEL
LIN {X 0,Y 420.629,Z 229.3,A -85,B 0,C 180,E1 -10020.461,E2 -10020.461} C_VEL
LIN {X 0,Y 420.37,Z 228.226,A -85,B 0,C 180,E1 -10020.517,E2 -10020.517} C_VEL
LIN {X 0,Y 418.847,Z 219.943,A -85,B 0,C 180,E1 -10022.474,E2 -10022.474} C_VEL
LIN {X 0,Y 418.292,Z 217.38,A -85,B 0,C 180,E1 -10023.099,E2 -10023.099} C_VEL
LIN {X 0,Y 418.244,Z 217.39,A -85,B 0,C 180,E1 -10026.237,E2 -10026.237} C_VEL
LIN {X 0,Y 418.257,Z 217.387,A -85,B 0,C 180,E1 -10029.679,E2 -10029.679} C_VEL
LIN {X 0,Y 418.237,Z 217.393,A -85,B 0,C 180,E1 -10032.322,E2 -10032.322} C_VEL
LIN {X 0,Y 418.24,Z 217.385,A -85,B 0,C 180,E1 -10035.109,E2 -10035.109} C_VEL
LIN {X 0,Y 418.279,Z 217.382,A -85,B 0,C 180,E1 -10037.771,E2 -10037.771} C_VEL
LIN {X 0,Y 418.25,Z 217.386,A -85,B 0,C 180,E1 -10041.558,E2 -10041.558} C_VEL
LIN {X 0,Y 418.243,Z 217.384,A -85,B 0,C 180,E1 -10045.157,E2 -10045.157} C_VEL
LIN {X 0,Y 418.227,Z 217.389,A -85,B 0,C 180,E1 -10047.47,E2 -10047.47} C_VEL
LIN {X 0,Y 418.256,Z 217.383,A -85,B 0,C 180,E1 -10050.892,E2 -10050.892} C_VEL
LIN {X 0,Y 418.249,Z 217.386,A -85,B 0,C 180,E1 -10054.094,E2 -10054.094} C_VEL
LIN {X 0,Y 418.21,Z 217.386,A -85,B 0,C 180,E1 -10057.262,E2 -10057.262} C_VEL
LIN {X 0,Y 418.258,Z 217.377,A -85,B 0,C 180,E1 -10060.363,E2 -10060.363} C_VEL
LIN {X 0,Y 418.3,Z 217.381,A -85,B 0,C 180,E1 -10063.404,E2 -10063.404} C_VEL
LIN {X 0,Y 418.32,Z 217.376,A -85,B 0,C 180,E1 -10066.999,E2 -10066.999} C_VEL
LIN {X 0,Y 418.313,Z 217.374,A -85,B 0,C 180,E1 -10070.328,E2 -10070.328} C_VEL
LIN {X 0,Y 418.471,Z 217.356,A -85,B 0,C 180,E1 -10073.248,E2 -10073.248} C_VEL
LIN {X 0,Y 418.311,Z 217.378,A -85,B 0,C 180,E1 -10075.181,E2 -10075.181} C_VEL
LIN {X 0,Y 418.51,Z 217.344,A -85,B 0,C 180,E1 -10078.075,E2 -10078.075} C_VEL
